  MoveL 6780 to (239.29, 155.73, 97.46) mm, rotated rx -180 ry 0 rz 180 deg; joints [-29.499, 18.299, 56.156, 64.652, 33.015, -60.536]
  Call Extruder(263.09151)
  MoveL 6781 to (239.16, 156.02, 97.46) mm, rotated rx 180 ry 0 rz -180 deg; joints [-29.531, 18.307, 56.146, 64.678, 33.044, -60.557]
  MoveL 6782 to (239.16, 156.02, 97.46) mm, rotated rx 180 ry 0 rz -180 deg; joints [-29.531, 18.307, 56.146, 64.678, 33.044, -60.557]
  Call Extruder(263.26194)
  MoveL 6783 to (239.05, 156.29, 97.46) mm, rotated rx 180 ry 0 rz 180 deg; joints [-29.561, 18.313, 56.137, 64.702, 33.071, -60.576]
  MoveL 6784 to (239.05, 156.29, 97.46) mm, rotated rx 180 ry 0 rz 180 deg; joints [-29.561, 18.313, 56.137, 64.702, 33.071, -60.576]
  Call Extruder(263.41995)
  MoveL 6785 to (238.94, 156.54, 97.46) mm, rotated rx -180 ry 0 rz 180 deg; joints [-29.589, 18.319, 56.129, 64.725, 33.096, -60.594]
  MoveL 6786 to (238.94, 156.54, 97.46) mm, rotated rx -180 ry 0 rz 180 deg; joints [-29.589, 18.319, 56.129, 64.725, 33.096, -60.594]
  Call Extruder(263.57856)
  MoveL 6787 to (238.84, 156.79, 97.46) mm, rotated rx 180 ry 0 rz 180 deg; joints [-29.617, 18.325, 56.121, 64.747, 33.121, -60.611]
  MoveL 6788 to (238.84, 156.79, 97.46) mm, rotated rx 180 ry 0 rz 180 deg; joints [-29.617, 18.325, 56.121, 64.747, 33.121, -60.611]
  Call Extruder(263.78473)
  MoveL 6789 to (238.66, 157.09, 97.46) mm, rotated rx -180 ry 0 rz 180 deg; joints [-29.653, 18.325, 56.121, 64.78, 33.153, -60.639]
  MoveL 6790 to (238.66, 157.09, 97.46) mm, rotated rx -180 ry 0 rz 180 deg; joints [-29.653, 18.325, 56.121, 64.78, 33.153, -60.639]
  Call Extruder(263.99168)
  MoveL 6791 to (238.49, 157.4, 97.46) mm, rotated rx 180 ry 0 rz 180 deg; joints [-29.689, 18.325, 56.122, 64.812, 33.184, -60.666]
  MoveL 6792 to (238.49, 157.4, 97.46) mm, rotated rx 180 ry 0 rz 180 deg; joints [-29.689, 18.325, 56.122, 64.812, 33.184, -60.666]
  Call Extruder(264.19941)
  MoveL 6793 to (238.31, 157.7, 97.46) mm, rotated rx -180 ry 0 rz -180 deg; joints [-29.725, 18.324, 56.122, 64.845, 33.216, -60.693]
  MoveL 6794 to (238.31, 157.7, 97.46) mm, rotated rx -180 ry 0 rz -180 deg; joints [-29.725, 18.324, 56.122, 64.845, 33.216, -60.693]
  Call Extruder(264.40791)
  MoveL 6795 to (238.13, 158.01, 97.46) mm, rotated rx 180 ry 0 rz 180 deg; joints [-29.761, 18.324, 56.123, 64.877, 33.247, -60.721]
  MoveL 6796 to (238.13, 158.01, 97.46) mm, rotated rx 180 ry 0 rz 180 deg; joints [-29.761, 18.324, 56.123, 64.877, 33.247, -60.721]
  Call Extruder(264.58745)
  MoveL 6797 to (237.96, 158.25, 97.46) mm, rotated rx 180 ry 0 rz 180 deg; joints [-29.792, 18.318, 56.131, 64.907, 33.273, -60.747]
  MoveL 6798 to (237.96, 158.25, 97.46) mm, rotated rx 180 ry 0 rz 180 deg; joints [-29.792, 18.318, 56.131, 64.907, 33.273, -60.747]
  Call Extruder(264.92086)
  MoveL 6799 to (237.63, 158.7, 97.46) mm, rotated rx -180 ry 0 rz 180 deg; joints [-29.849, 18.306, 56.147, 64.963, 33.322, -60.796]
  MoveL 6800 to (237.63, 158.7, 97.46) mm, rotated rx -180 ry 0 rz 180 deg; joints [-29.849, 18.306, 56.147, 64.963, 33.322, -60.796]
  Call Extruder(265.25545)
  MoveL 6801 to (237.3, 159.15, 97.46) mm, rotated rx 180 ry 0 rz 180 deg; joints [-29.907, 18.294, 56.162, 65.019, 33.37, -60.844]
  Call Extruder(266.08341)
  MoveL 6802 to (236.39, 160.19, 97.46) mm, rotated rx 180 ry 0 rz -180 deg; joints [-30.046, 18.239, 56.234, 65.166, 33.485, -60.975]
  Call Extruder(266.91134)
  MoveL 6803 to (235.35, 161.1, 97.46) mm, rotated rx 180 ry 0 rz 180 deg; joints [-30.182, 18.151, 56.349, 65.322, 33.592, -61.119]
  Call Extruder(267.07865)
  MoveL 6804 to (235.13, 161.27, 97.46) mm, rotated rx 180 ry 0 rz 180 deg; joints [-30.208, 18.129, 56.379, 65.355, 33.612, -61.15]
  MoveL 6805 to (235.13, 161.27, 97.46) mm, rotated rx 180 ry 0 rz 180 deg; joints [-30.208, 18.129, 56.379, 65.355, 33.612, -61.15]
  Call Extruder(267.41207)
  MoveL 6806 to (234.68, 161.59, 97.46) mm, rotated rx 180 ry 0 rz 180 deg; joints [-30.261, 18.084, 56.438, 65.419, 33.652, -61.211]
  MoveL 6807 to (234.68, 161.59, 97.46) mm, rotated rx 180 ry 0 rz 180 deg; joints [-30.261, 18.084, 56.438, 65.419, 33.652, -61.211]
  Call Extruder(267.74432)
  MoveL 6808 to (234.23, 161.92, 97.46) mm, rotated rx 180 ry 0 rz 180 deg; joints [-30.314, 18.039, 56.497, 65.484, 33.693, -61.271]
  MoveL 6809 to (234.23, 161.92, 97.46) mm, rotated rx 180 ry 0 rz 180 deg; joints [-30.314, 18.039, 56.497, 65.484, 33.693, -61.271]
  Call Extruder(267.86197)
  MoveL 6810 to (234.05, 162.02, 97.46) mm, rotated rx 180 ry 0 rz 180 deg; joints [-30.331, 18.019, 56.522, 65.508, 33.706, -61.294]
  MoveL 6811 to (234.05, 162.02, 97.46) mm, rotated rx 180 ry 0 rz 180 deg; joints [-30.331, 18.019, 56.522, 65.508, 33.706, -61.294]
  Call Extruder(268.06970)
  MoveL 6812 to (233.75, 162.2, 97.46) mm, rotated rx 180 ry 0 rz 180 deg; joints [-30.363, 17.985, 56.567, 65.55, 33.729, -61.334]
  MoveL 6813 to (233.75, 162.2, 97.46) mm, rotated rx 180 ry 0 rz 180 deg; joints [-30.363, 17.985, 56.567, 65.55, 33.729, -61.334]
  Call Extruder(268.27665)
  MoveL 6814 to (233.45, 162.37, 97.46) mm, rotated rx 180 ry 0 rz 180 deg; joints [-30.394, 17.95, 56.613, 65.591, 33.753, -61.374]
  MoveL 6815 to (233.45, 162.37, 97.46) mm, rotated rx 180 ry 0 rz 180 deg; joints [-30.394, 17.95, 56.613, 65.591, 33.753, -61.374]
  Call Extruder(268.48282)
  MoveL 6816 to (233.14, 162.55, 97.46) mm, rotated rx 180 ry 0 rz 180 deg; joints [-30.426, 17.916, 56.658, 65.633, 33.776, -61.414]
  MoveL 6817 to (233.14, 162.55, 97.46) mm, rotated rx 180 ry 0 rz 180 deg; joints [-30.426, 17.916, 56.658, 65.633, 33.776, -61.414]
  Call Extruder(268.66449)
  MoveL 6818 to (232.87, 162.69, 97.46) mm, rotated rx -180 ry 0 rz 180 deg; joints [-30.453, 17.882, 56.701, 65.67, 33.796, -61.45]
  MoveL 6819 to (232.87, 162.69, 97.46) mm, rotated rx -180 ry 0 rz 180 deg; joints [-30.453, 17.882, 56.701, 65.67, 33.796, -61.45]
  Call Extruder(268.82246)
  MoveL 6820 to (232.62, 162.8, 97.46) mm, rotated rx -180 ry 0 rz 180 deg; joints [-30.476, 17.85, 56.743, 65.703, 33.811, -61.483]
  MoveL 6821 to (232.62, 162.8, 97.46) mm, rotated rx -180 ry 0 rz 180 deg; joints [-30.476, 17.85, 56.743, 65.703, 33.811, -61.483]
  Call Extruder(268.97983)
  MoveL 6822 to (232.37, 162.9, 97.46) mm, rotated rx 180 ry 0 rz 180 deg; joints [-30.498, 17.819, 56.784, 65.736, 33.827, -61.515]
  MoveL 6823 to (232.37, 162.9, 97.46) mm, rotated rx 180 ry 0 rz 180 deg; joints [-30.498, 17.819, 56.784, 65.736, 33.827, -61.515]
  Call Extruder(269.16257)
  MoveL 6824 to (232.08, 163.02, 97.46) mm, rotated rx 180 ry 0 rz 180 deg; joints [-30.524, 17.781, 56.834, 65.774, 33.846, -61.552]
  MoveL 6825 to (232.08, 163.02, 97.46) mm, rotated rx 180 ry 0 rz 180 deg; joints [-30.524, 17.781, 56.834, 65.774, 33.846, -61.552]
  Call Extruder(269.34456)
  MoveL 6826 to (231.78, 163.15, 97.46) mm, rotated rx -180 ry 0 rz 180 deg; joints [-30.551, 17.743, 56.883, 65.812, 33.864, -61.589]
  MoveL 6827 to (231.78, 163.15, 97.46) mm, rotated rx -180 ry 0 rz 180 deg; joints [-30.551, 17.743, 56.883, 65.812, 33.864, -61.589]
  Call Extruder(269.49190)
  MoveL 6828 to (231.54, 163.24, 97.46) mm, rotated rx 180 ry 0 rz 180 deg; joints [-30.571, 17.711, 56.924, 65.842, 33.878, -61.62]
  MoveL 6829 to (231.54, 163.24, 97.46) mm, rotated rx 180 ry 0 rz 180 deg; joints [-30.571, 17.711, 56.924, 65.842, 33.878, -61.62]
  Call Extruder(269.60512)
  MoveL 6830 to (231.35, 163.3, 97.46) mm, rotated rx 180 ry 0 rz 180 deg; joints [-30.587, 17.685, 56.958, 65.866, 33.889, -61.644]
  MoveL 6831 to (231.35, 163.3, 97.46) mm, rotated rx 180 ry 0 rz 180 deg; joints [-30.587, 17.685, 56.958, 65.866, 33.889, -61.644]
  Call Extruder(269.71789)
  MoveL 6832 to (231.17, 163.36, 97.46) mm, rotated rx 180 ry 0 rz 180 deg; joints [-30.602, 17.659, 56.992, 65.89, 33.899, -61.667]
  MoveL 6833 to (231.17, 163.36, 97.46) mm, rotated rx 180 ry 0 rz 180 deg; joints [-30.602, 17.659, 56.992, 65.89, 33.899, -61.667]
  Call Extruder(269.83022)
  MoveL 6834 to (230.98, 163.42, 97.46) mm, rotated rx 180 ry 0 rz -180 deg; joints [-30.618, 17.633, 57.026, 65.914, 33.909, -61.691]
  MoveL 6835 to (230.98, 163.42, 97.46) mm, rotated rx 180 ry 0 rz -180 deg; joints [-30.618, 17.633, 57.026, 65.914, 33.909, -61.691]
  Call Extruder(269.94211)
  MoveL 6836 to (230.79, 163.48, 97.46) mm, rotated rx 180 ry 0 rz 180 deg; joints [-30.633, 17.607, 57.06, 65.937, 33.92, -61.715]
  MoveL 6837 to (230.79, 163.48, 97.46) mm, rotated rx 180 ry 0 rz 180 deg; joints [-30.633, 17.607, 57.06, 65.937, 33.92, -61.715]
  Call Extruder(270.06351)
  MoveL 6838 to (230.58, 163.55, 97.46) mm, rotated rx 180 ry 0 rz 180 deg; joints [-30.65, 17.579, 57.097, 65.963, 33.931, -61.74]
  MoveL 6839 to (230.58, 163.55, 97.46) mm, rotated rx 180 ry 0 rz 180 deg; joints [-30.65, 17.579, 57.097, 65.963, 33.931, -61.74]
  Call Extruder(270.19433)
  MoveL 6840 to (230.36, 163.62, 97.46) mm, rotated rx 180 ry 0 rz 180 deg; joints [-30.668, 17.548, 57.137, 65.991, 33.943, -61.768]
  MoveL 6841 to (230.36, 163.62, 97.46) mm, rotated rx 180 ry 0 rz 180 deg; joints [-30.668, 17.548, 57.137, 65.991, 33.943, -61.768]
  Call Extruder(270.32458)
  MoveL 6842 to (230.14, 163.68, 97.46) mm, rotated rx 180 ry 0 rz 180 deg; joints [-30.685, 17.516, 57.178, 66.019, 33.955, -61.796]
  MoveL 6843 to (230.14, 163.68, 97.46) mm, rotated rx 180 ry 0 rz 180 deg; joints [-30.685, 17.516, 57.178, 66.019, 33.955, -61.796]
  Call Extruder(270.45426)
  MoveL 6844 to (229.91, 163.75, 97.46) mm, rotated rx 180 ry 0 rz 180 deg; joints [-30.703, 17.485, 57.218, 66.047, 33.967, -61.824]
  MoveL 6845 to (229.91, 163.75, 97.46) mm, rotated rx 180 ry 0 rz 180 deg; joints [-30.703, 17.485, 57.218, 66.047, 33.967, -61.824]
  Call Extruder(270.58338)
  MoveL 6846 to (229.69, 163.82, 97.46) mm, rotated rx -180 ry 0 rz -180 deg; joints [-30.721, 17.454, 57.259, 66.074, 33.979, -61.852]
  MoveL 6847 to (229.69, 163.82, 97.46) mm, rotated rx -180 ry 0 rz -180 deg; joints [-30.721, 17.454, 57.259, 66.074, 33.979, -61.852]
  Call Extruder(270.69845)
  MoveL 6848 to (229.48, 163.86, 97.46) mm, rotated rx -180 ry 0 rz -180 deg; joints [-30.736, 17.424, 57.298, 66.099, 33.988, -61.877]
  MoveL 6849 to (229.48, 163.86, 97.46) mm, rotated rx -180 ry 0 rz -180 deg; joints [-30.736, 17.424, 57.298, 66.099, 33.988, -61.877]
  Call Extruder(270.81308)
  MoveL 6850 to (229.28, 163.91, 97.46) mm, rotated rx 180 ry 0 rz 180 deg; joints [-30.751, 17.394, 57.337, 66.124, 33.998, -61.902]
  MoveL 6851 to (229.28, 163.91, 97.46) mm, rotated rx 180 ry 0 rz 180 deg; joints [-30.751, 17.394, 57.337, 66.124, 33.998, -61.902]
  Call Extruder(270.92725)
  MoveL 6852 to (229.08, 163.95, 97.46) mm, rotated rx 180 ry 0 rz 180 deg; joints [-30.766, 17.364, 57.376, 66.148, 34.007, -61.927]
  MoveL 6853 to (229.08, 163.95, 97.46) mm, rotated rx 180 ry 0 rz 180 deg; joints [-30.766, 17.364, 57.376, 66.148, 34.007, -61.927]
  Call Extruder(271.04096)
  MoveL 6854 to (228.87, 164, 97.46) mm, rotated rx -180 ry 0 rz 180 deg; joints [-30.781, 17.334, 57.415, 66.173, 34.017, -61.952]
  MoveL 6855 to (228.87, 164, 97.46) mm, rotated rx -180 ry 0 rz 180 deg; joints [-30.781, 17.334, 57.415, 66.173, 34.017, -61.952]
  Call Extruder(271.16638)
  MoveL 6856 to (228.64, 164.04, 97.46) mm, rotated rx -180 ry 0 rz 180 deg; joints [-30.797, 17.3, 57.458, 66.2, 34.027, -61.979]
  MoveL 6857 to (228.64, 164.04, 97.46) mm, rotated rx -180 ry 0 rz 180 deg; joints [-30.797, 17.3, 57.458, 66.2, 34.027, -61.979]
  Call Extruder(271.30336)
  MoveL 6858 to (228.4, 164.09, 97.46) mm, rotated rx 180 ry 0 rz 180 deg; joints [-30.815, 17.263, 57.506, 66.23, 34.038, -62.01]
  MoveL 6859 to (228.4, 164.09, 97.46) mm, rotated rx 180 ry 0 rz 180 deg; joints [-30.815, 17.263, 57.506, 66.23, 34.038, -62.01]
  Call Extruder(271.43973)
  MoveL 6860 to (228.15, 164.14, 97.46) mm, rotated rx 180 ry 0 rz 180 deg; joints [-30.832, 17.226, 57.555, 66.259, 34.05, -62.04]
  MoveL 6861 to (228.15, 164.14, 97.46) mm, rotated rx 180 ry 0 rz 180 deg; joints [-30.832, 17.226, 57.555, 66.259, 34.05, -62.04]
  Call Extruder(271.57549)
  MoveL 6862 to (227.9, 164.19, 97.46) mm, rotated rx -180 ry 0 rz 180 deg; joints [-30.85, 17.189, 57.602, 66.289, 34.061, -62.07]
  MoveL 6863 to (227.9, 164.19, 97.46) mm, rotated rx -180 ry 0 rz 180 deg; joints [-30.85, 17.189, 57.602, 66.289, 34.061, -62.07]
  Call Extruder(271.71064)
  MoveL 6864 to (227.65, 164.24, 97.46) mm, rotated rx 180 ry 0 rz 180 deg; joints [-30.868, 17.152, 57.65, 66.319, 34.072, -62.1]
  MoveL 6865 to (227.65, 164.24, 97.46) mm, rotated rx 180 ry 0 rz 180 deg; joints [-30.868, 17.152, 57.65, 66.319, 34.072, -62.1]
  Call Extruder(271.84517)
  MoveL 6866 to (227.4, 164.29, 97.46) mm, rotated rx 180 ry 0 rz 180 deg; joints [-30.886, 17.115, 57.698, 66.348, 34.083, -62.13]
  MoveL 6867 to (227.4, 164.29, 97.46) mm, rotated rx 180 ry 0 rz 180 deg; joints [-30.886, 17.115, 57.698, 66.348, 34.083, -62.13]
  Call Extruder(271.97910)
  MoveL 6868 to (227.15, 164.34, 97.46) mm, rotated rx 180 ry 0 rz 180 deg; joints [-30.903, 17.078, 57.746, 66.377, 34.095, -62.16]
  MoveL 6869 to (227.15, 164.34, 97.46) mm, rotated rx 180 ry 0 rz 180 deg; joints [-30.903, 17.078, 57.746, 66.377, 34.095, -62.16]
  Call Extruder(272.12696)
  MoveL 6870 to (226.87, 164.39, 97.46) mm, rotated rx 180 ry 0 rz 180 deg; joints [-30.923, 17.037, 57.799, 66.41, 34.107, -62.193]
  MoveL 6871 to (226.87, 164.39, 97.46) mm, rotated rx 180 ry 0 rz 180 deg; joints [-30.923, 17.037, 57.799, 66.41, 34.107, -62.193]
  Call Extruder(272.28870)
  MoveL 6872 to (226.57, 164.44, 97.46) mm, rotated rx 180 ry 0 rz 180 deg; joints [-30.943, 16.99, 57.859, 66.445, 34.12, -62.229]
  MoveL 6873 to (226.57, 164.44, 97.46) mm, rotated rx 180 ry 0 rz 180 deg; joints [-30.943, 16.99, 57.859, 66.445, 34.12, -62.229]
  Call Extruder(272.44972)
  MoveL 6874 to (226.26, 164.49, 97.46) mm, rotated rx 180 ry 0 rz 180 deg; joints [-30.964, 16.944, 57.919, 66.481, 34.133, -62.265]
  MoveL 6875 to (226.26, 164.49, 97.46) mm, rotated rx 180 ry 0 rz 180 deg; joints [-30.964, 16.944, 57.919, 66.481, 34.133, -62.265]
  Call Extruder(272.61000)
  MoveL 6876 to (225.96, 164.54, 97.46) mm, rotated rx 180 ry 0 rz 180 deg; joints [-30.985, 16.897, 57.979, 66.516, 34.146, -62.301]
  MoveL 6877 to (225.96, 164.54, 97.46) mm, rotated rx 180 ry 0 rz 180 deg; joints [-30.985, 16.897, 57.979, 66.516, 34.146, -62.301]
  Call Extruder(272.76956)
  MoveL 6878 to (225.65, 164.58, 97.46) mm, rotated rx 180 ry 0 rz 180 deg; joints [-31.006, 16.851, 58.038, 66.551, 34.159, -62.337]
  MoveL 6879 to (225.65, 164.58, 97.46) mm, rotated rx 180 ry 0 rz 180 deg; joints [-31.006, 16.851, 58.038, 66.551, 34.159, -62.337]
  Call Extruder(272.92838)
  MoveL 6880 to (225.34, 164.63, 97.46) mm, rotated rx 180 ry 0 rz 180 deg; joints [-31.027, 16.805, 58.098, 66.586, 34.172, -62.373]
  MoveL 6881 to (225.34, 164.63, 97.46) mm, rotated rx 180 ry 0 rz 180 deg; joints [-31.027, 16.805, 58.098, 66.586, 34.172, -62.373]
  Call Extruder(273.10706)
  MoveL 6882 to (225, 164.68, 97.46) mm, rotated rx 180 ry 0 rz 180 deg; joints [-31.049, 16.752, 58.166, 66.626, 34.187, -62.414]
  MoveL 6883 to (225, 164.68, 97.46) mm, rotated rx 180 ry 0 rz 180 deg; joints [-31.049, 16.752, 58.166, 66.626, 34.187, -62.414]
  Call Extruder(273.30550)
  MoveL 6884 to (224.61, 164.73, 97.46) mm, rotated rx -180 ry 0 rz -180 deg; joints [-31.074, 16.692, 58.243, 66.67, 34.202, -62.459]
  MoveL 6885 to (224.61, 164.73, 97.46) mm, rotated rx -180 ry 0 rz -180 deg; joints [-31.074, 16.692, 58.243, 66.67, 34.202, -62.459]
  Call Extruder(273.50307)
  MoveL 6886 to (224.22, 164.77, 97.46) mm, rotated rx 180 ry 0 rz 180 deg; joints [-31.1, 16.632, 58.32, 66.713, 34.217, -62.504]
  MoveL 6887 to (224.22, 164.77, 97.46) mm, rotated rx 180 ry 0 rz 180 deg; joints [-31.1, 16.632, 58.32, 66.713, 34.217, -62.504]
  Call Extruder(273.69978)
  MoveL 6888 to (223.84, 164.82, 97.46) mm, rotated rx 180 ry 0 rz 180 deg; joints [-31.125, 16.573, 58.397, 66.757, 34.233, -62.548]
  MoveL 6889 to (223.84, 164.82, 97.46) mm, rotated rx 180 ry 0 rz 180 deg; joints [-31.125, 16.573, 58.397, 66.757, 34.233, -62.548]
  Call Extruder(273.89562)
  MoveL 6890 to (223.45, 164.86, 97.46) mm, rotated rx 180 ry 0 rz 180 deg; joints [-31.15, 16.513, 58.473, 66.8, 34.249, -62.593]
  MoveL 6891 to (223.45, 164.86, 97.46) mm, rotated rx 180 ry 0 rz 180 deg; joints [-31.15, 16.513, 58.473, 66.8, 34.249, -62.593]
  Call Extruder(274.19098)
  MoveL 6892 to (222.86, 164.91, 97.46) mm, rotated rx -180 ry 0 rz 180 deg; joints [-31.186, 16.42, 58.592, 66.865, 34.27, -62.66]
  MoveL 6893 to (222.86, 164.91, 97.46) mm, rotated rx -180 ry 0 rz 180 deg; joints [-31.186, 16.42, 58.592, 66.865, 34.27, -62.66]
  Call Extruder(274.48500)
  MoveL 6894 to (222.27, 164.95, 97.46) mm, rotated rx -180 ry 0 rz 180 deg; joints [-31.222, 16.327, 58.711, 66.929, 34.292, -62.727]
  MoveL 6895 to (222.27, 164.95, 97.46) mm, rotated rx -180 ry 0 rz 180 deg; joints [-31.222, 16.327, 58.711, 66.929, 34.292, -62.727]
  Call Extruder(274.77770)
  MoveL 6896 to (221.68, 165, 97.46) mm, rotated rx 180 ry 0 rz 180 deg; joints [-31.258, 16.235, 58.829, 66.993, 34.315, -62.793]
  MoveL 6897 to (221.68, 165, 97.46) mm, rotated rx 180 ry 0 rz 180 deg; joints [-31.258, 16.235, 58.829, 66.993, 34.315, -62.793]
  Call Extruder(275.35114)
  MoveL 6898 to (220.52, 165.05, 97.46) mm, rotated rx 180 ry 0 rz 180 deg; joints [-31.326, 16.048, 59.067, 67.117, 34.355, -62.922]
  MoveL 6899 to (220.52, 165.05, 97.46) mm, rotated rx 180 ry 0 rz 180 deg; joints [-31.326, 16.048, 59.067, 67.117, 34.355, -62.922]
  Call Extruder(276.06515)
  MoveL 6900 to (219.06, 165.09, 97.46) mm, rotated rx 180 ry 0 rz 180 deg; joints [-31.409, 15.814, 59.365, 67.27, 34.404, -63.081]
  Call Extruder(392.91189)
  MoveL 6901 to (-19.06, 165.09, 97.46) mm, rotated rx 180 ry 0 rz 180 deg; joints [-51.475, -13.284, 89.091, 78.954, 52.855, -72.085]
  Call Extruder(393.34049)
  MoveL 6902 to (-19.94, 165.07, 97.46) mm, rotated rx -180 ry 0 rz 180 deg; joints [-51.582, -13.365, 89.153, 78.982, 52.96, -72.087]
  MoveL 6903 to (-19.94, 165.07, 97.46) mm, rotated rx -180 ry 0 rz 180 deg; joints [-51.582, -13.365, 89.153, 78.982, 52.96, -72.087]
  Call Extruder(393.91395)
  MoveL 6904 to (-21.1, 165.03, 97.46) mm, rotated rx 180 ry 0 rz -180 deg; joints [-51.722, -13.474, 89.237, 79.017, 53.098, -72.089]
  MoveL 6905 to (-21.1, 165.03, 97.46) mm, rotated rx 180 ry 0 rz -180 deg; joints [-51.722, -13.474, 89.237, 79.017, 53.098, -72.089]
  Call Extruder(394.34824)
  MoveL 6906 to (-21.97, 164.98, 97.46) mm, rotated rx 180 ry 0 rz 180 deg; joints [-51.827, -13.557, 89.301, 79.044, 53.201, -72.09]
  MoveL 6907 to (-21.97, 164.98, 97.46) mm, rotated rx 180 ry 0 rz 180 deg; joints [-51.827, -13.557, 89.301, 79.044, 53.201, -72.09]
  Call Extruder(394.64227)
  MoveL 6908 to (-22.56, 164.93, 97.46) mm, rotated rx 180 ry 0 rz -180 deg; joints [-51.897, -13.615, 89.345, 79.06, 53.27, -72.089]
  MoveL 6909 to (-22.56, 164.93, 97.46) mm, rotated rx 180 ry 0 rz -180 deg; joints [-51.897, -13.615, 89.345, 79.06, 53.27, -72.089]
  Call Extruder(394.93763)
  MoveL 6910 to (-23.15, 164.89, 97.46) mm, rotated rx 180 ry 0 rz 180 deg; joints [-51.966, -13.672, 89.39, 79.077, 53.339, -72.089]
  MoveL 6911 to (-23.15, 164.89, 97.46) mm, rotated rx 180 ry 0 rz 180 deg; joints [-51.966, -13.672, 89.39, 79.077, 53.339, -72.089]
  Call Extruder(395.18385)
  MoveL 6912 to (-23.64, 164.84, 97.46) mm, rotated rx 180 ry 0 rz 180 deg; joints [-52.023, -13.721, 89.427, 79.091, 53.395, -72.088]
  MoveL 6913 to (-23.64, 164.84, 97.46) mm, rotated rx 180 ry 0 rz 180 deg; joints [-52.023, -13.721, 89.427, 79.091, 53.395, -72.088]
  Call Extruder(395.38056)
  MoveL 6914 to (-24.03, 164.79, 97.46) mm, rotated rx 180 ry 0 rz 180 deg; joints [-52.067, -13.76, 89.457, 79.101, 53.439, -72.087]
  MoveL 6915 to (-24.03, 164.79, 97.46) mm, rotated rx 180 ry 0 rz 180 deg; joints [-52.067, -13.76, 89.457, 79.101, 53.439, -72.087]
  Call Extruder(395.57813)
  MoveL 6916 to (-24.42, 164.75, 97.46) mm, rotated rx -180 ry 0 rz 180 deg; joints [-52.112, -13.8, 89.487, 79.111, 53.483, -72.085]
  MoveL 6917 to (-24.42, 164.75, 97.46) mm, rotated rx -180 ry 0 rz 180 deg; joints [-52.112, -13.8, 89.487, 79.111, 53.483, -72.085]
  Call Extruder(395.77657)
  MoveL 6918 to (-24.8, 164.7, 97.46) mm, rotated rx -180 ry 0 rz 180 deg; joints [-52.156, -13.839, 89.517, 79.121, 53.527, -72.084]
  MoveL 6919 to (-24.8, 164.7, 97.46) mm, rotated rx -180 ry 0 rz 180 deg; joints [-52.156, -13.839, 89.517, 79.121, 53.527, -72.084]
  Call Extruder(395.97588)
  MoveL 6920 to (-25.19, 164.66, 97.46) mm, rotated rx 180 ry 0 rz 180 deg; joints [-52.2, -13.878, 89.547, 79.132, 53.571, -72.083]
  MoveL 6921 to (-25.19, 164.66, 97.46) mm, rotated rx 180 ry 0 rz 180 deg; joints [-52.2, -13.878, 89.547, 79.132, 53.571, -72.083]
  Call Extruder(396.13471)
  MoveL 6922 to (-25.5, 164.61, 97.46) mm, rotated rx 180 ry 0 rz 180 deg; joints [-52.235, -13.911, 89.572, 79.139, 53.605, -72.081]
  MoveL 6923 to (-25.5, 164.61, 97.46) mm, rotated rx 180 ry 0 rz 180 deg; joints [-52.235, -13.911, 89.572, 79.139, 53.605, -72.081]
  Call Extruder(396.29427)
  MoveL 6924 to (-25.8, 164.56, 97.46) mm, rotated rx 180 ry 0 rz 180 deg; joints [-52.269, -13.943, 89.597, 79.147, 53.639, -72.08]
  MoveL 6925 to (-25.8, 164.56, 97.46) mm, rotated rx 180 ry 0 rz 180 deg; joints [-52.269, -13.943, 89.597, 79.147, 53.639, -72.08]
  Call Extruder(396.45456)
  MoveL 6926 to (-26.11, 164.51, 97.46) mm, rotated rx 180 ry 0 rz -180 deg; joints [-52.303, -13.976, 89.621, 79.154, 53.672, -72.078]
  MoveL 6927 to (-26.11, 164.51, 97.46) mm, rotated rx 180 ry 0 rz -180 deg; joints [-52.303, -13.976, 89.621, 79.154, 53.672, -72.078]
  Call Extruder(396.61557)
  MoveL 6928 to (-26.41, 164.46, 97.46) mm, rotated rx 180 ry 0 rz -180 deg; joints [-52.337, -14.008, 89.646, 79.161, 53.706, -72.076]
  MoveL 6929 to (-26.41, 164.46, 97.46) mm, rotated rx 180 ry 0 rz -180 deg; joints [-52.337, -14.008, 89.646, 79.161, 53.706, -72.076]
  Call Extruder(396.77732)
  MoveL 6930 to (-26.72, 164.41, 97.46) mm, rotated rx 180 ry 0 rz 180 deg; joints [-52.371, -14.04, 89.671, 79.169, 53.74, -72.075]
  MoveL 6931 to (-26.72, 164.41, 97.46) mm, rotated rx 180 ry 0 rz 180 deg; joints [-52.371, -14.04, 89.671, 79.169, 53.74, -72.075]
  Call Extruder(396.93979)
  MoveL 6932 to (-27.02, 164.37, 97.46) mm, rotated rx 180 ry 0 rz 180 deg; joints [-52.405, -14.073, 89.695, 79.176, 53.774, -72.073]
  MoveL 6933 to (-27.02, 164.37, 97.46) mm, rotated rx 180 ry 0 rz 180 deg; joints [-52.405, -14.073, 89.695, 79.176, 53.774, -72.073]
  Call Extruder(397.07371)
  MoveL 6934 to (-27.27, 164.32, 97.46) mm, rotated rx -180 ry 0 rz -180 deg; joints [-52.432, -14.1, 89.716, 79.182, 53.801, -72.071]
  MoveL 6935 to (-27.27, 164.32, 97.46) mm, rotated rx -180 ry 0 rz -180 deg; joints [-52.432, -14.1, 89.716, 79.182, 53.801, -72.071]
  Call Extruder(397.20825)
  MoveL 6936 to (-27.52, 164.27, 97.46) mm, rotated rx 180 ry 0 rz 180 deg; joints [-52.459, -14.127, 89.737, 79.187, 53.828, -72.069]
  MoveL 6937 to (-27.52, 164.27, 97.46) mm, rotated rx 180 ry 0 rz 180 deg; joints [-52.459, -14.127, 89.737, 79.187, 53.828, -72.069]
  Call Extruder(397.34340)
  MoveL 6938 to (-27.77, 164.22, 97.46) mm, rotated rx 180 ry 0 rz 180 deg; joints [-52.486, -14.155, 89.758, 79.193, 53.855, -72.067]
  MoveL 6939 to (-27.77, 164.22, 97.46) mm, rotated rx 180 ry 0 rz 180 deg; joints [-52.486, -14.155, 89.758, 79.193, 53.855, -72.067]
  Call Extruder(397.47915)
  MoveL 6940 to (-28.02, 164.17, 97.46) mm, rotated rx 180 ry 0 rz -180 deg; joints [-52.513, -14.182, 89.779, 79.199, 53.882, -72.065]
  MoveL 6941 to (-28.02, 164.17, 97.46) mm, rotated rx 180 ry 0 rz -180 deg; joints [-52.513, -14.182, 89.779, 79.199, 53.882, -72.065]
  Call Extruder(397.61552)
  MoveL 6942 to (-28.27, 164.12, 97.46) mm, rotated rx 180 ry 0 rz 180 deg; joints [-52.54, -14.21, 89.799, 79.204, 53.909, -72.063]
  MoveL 6943 to (-28.27, 164.12, 97.46) mm, rotated rx 180 ry 0 rz 180 deg; joints [-52.54, -14.21, 89.799, 79.204, 53.909, -72.063]
  Call Extruder(397.70039)
  MoveL 6944 to (-28.43, 164.09, 97.46) mm, rotated rx 180 ry 0 rz -180 deg; joints [-52.556, -14.227, 89.812, 79.208, 53.925, -72.062]
  Set speed (130.0 mm/s)
  MoveL 6945 to (-31.76, 163.31, 97.46) mm, rotated rx 180 ry 0 rz 180 deg; joints [-52.91, -14.605, 90.097, 79.276, 54.279, -72.028]
  MoveL 6946 to (-31.76, 163.31, 106.87) mm, rotated rx 180 ry 0 rz 180 deg; joints [-52.91, -15.274, 92.047, 80.186, 54.05, -73.582]
  Call Extruder(395.70039)
  Set speed (40.0 mm/s)
  MoveL 6947 to (-31.76, 163.31, 106.87) mm, rotated rx 180 ry 0 rz 180 deg; joints [-52.91, -15.274, 92.047, 80.186, 54.05, -73.582]
  Call Extruder(0.00000)
  Set speed (130.0 mm/s)
  MoveL 6948 to (-31.64, 163.21, 106.87) mm, rotated rx 180 ry 0 rz 180 deg; joints [-52.884, -15.275, 92.048, 80.177, 54.026, -73.576]
  Call Extruder(2.00000)
  Set speed (40.0 mm/s)
  MoveL 6949 to (-31.64, 163.21, 106.87) mm, rotated rx 180 ry 0 rz 180 deg; joints [-52.884, -15.275, 92.048, 80.177, 54.026, -73.576]
  Set speed (30.0 mm/s)
  MoveL 6950 to (-31.64, 163.21, 106.87) mm, rotated rx 180 ry 0 rz 180 deg; joints [-52.884, -15.275, 92.048, 80.177, 54.026, -73.576]
  Call Extruder(2.18198)
  MoveL 6951 to (-31.93, 163.09, 106.87) mm, rotated rx 180 ry 0 rz 180 deg; joints [-52.91, -15.315, 92.077, 80.179, 54.052, -73.57]
  MoveL 6952 to (-31.93, 163.09, 106.87) mm, rotated rx 180 ry 0 rz 180 deg; joints [-52.91, -15.315, 92.077, 80.179, 54.052, -73.57]
  Call Extruder(2.36471)
  MoveL 6953 to (-32.22, 162.97, 106.87) mm, rotated rx -180 ry 0 rz -180 deg; joints [-52.936, -15.354, 92.106, 80.18, 54.079, -73.563]
  MoveL 6954 to (-32.22, 162.97, 106.87) mm, rotated rx -180 ry 0 rz -180 deg; joints [-52.936, -15.354, 92.106, 80.18, 54.079, -73.563]
  Call Extruder(2.53513)
  MoveL 6955 to (-32.49, 162.85, 106.87) mm, rotated rx 180 ry 0 rz 180 deg; joints [-52.96, -15.39, 92.133, 80.182, 54.104, -73.556]
  MoveL 6956 to (-32.49, 162.85, 106.87) mm, rotated rx 180 ry 0 rz 180 deg; joints [-52.96, -15.39, 92.133, 80.182, 54.104, -73.556]
  Call Extruder(2.69310)
  MoveL 6957 to (-32.74, 162.74, 106.87) mm, rotated rx -180 ry 0 rz 180 deg; joints [-52.982, -15.424, 92.159, 80.183, 54.126, -73.55]
  MoveL 6958 to (-32.74, 162.74, 106.87) mm, rotated rx -180 ry 0 rz 180 deg; joints [-52.982, -15.424, 92.159, 80.183, 54.126, -73.55]
  Call Extruder(2.85168)
  MoveL 6959 to (-32.99, 162.64, 106.87) mm, rotated rx 180 ry 0 rz -180 deg; joints [-53.004, -15.458, 92.184, 80.185, 54.149, -73.544]
  MoveL 6960 to (-32.99, 162.64, 106.87) mm, rotated rx 180 ry 0 rz -180 deg; joints [-53.004, -15.458, 92.184, 80.185, 54.149, -73.544]
  Call Extruder(3.05785)
  MoveL 6961 to (-33.29, 162.46, 106.87) mm, rotated rx 180 ry 0 rz 180 deg; joints [-53.026, -15.504, 92.218, 80.184, 54.172, -73.533]
  MoveL 6962 to (-33.29, 162.46, 106.87) mm, rotated rx 180 ry 0 rz 180 deg; joints [-53.026, -15.504, 92.218, 80.184, 54.172, -73.533]
  Call Extruder(3.26479)
  MoveL 6963 to (-33.6, 162.29, 106.87) mm, rotated rx -180 ry 0 rz 180 deg; joints [-53.049, -15.551, 92.252, 80.183, 54.196, -73.523]
  MoveL 6964 to (-33.6, 162.29, 106.87) mm, rotated rx -180 ry 0 rz 180 deg; joints [-53.049, -15.551, 92.252, 80.183, 54.196, -73.523]
  Call Extruder(3.47251)
  MoveL 6965 to (-33.9, 162.11, 106.87) mm, rotated rx 180 ry 0 rz 180 deg; joints [-53.071, -15.597, 92.286, 80.183, 54.22, -73.513]
  MoveL 6966 to (-33.9, 162.11, 106.87) mm, rotated rx 180 ry 0 rz 180 deg; joints [-53.071, -15.597, 92.286, 80.183, 54.22, -73.513]
  Call Extruder(3.68101)
  MoveL 6967 to (-34.21, 161.94, 106.87) mm, rotated rx 180 ry 0 rz 180 deg; joints [-53.094, -15.644, 92.32, 80.182, 54.243, -73.503]
  MoveL 6968 to (-34.21, 161.94, 106.87) mm, rotated rx 180 ry 0 rz 180 deg; joints [-53.094, -15.644, 92.32, 80.182, 54.243, -73.503]
  Call Extruder(3.86055)
  MoveL 6969 to (-34.45, 161.76, 106.87) mm, rotated rx -180 ry 0 rz 180 deg; joints [-53.109, -15.685, 92.351, 80.179, 54.259, -73.493]
  MoveL 6970 to (-34.45, 161.76, 106.87) mm, rotated rx -180 ry 0 rz 180 deg; joints [-53.109, -15.685, 92.351, 80.179, 54.259, -73.493]
  Call Extruder(4.19399)
  MoveL 6971 to (-34.9, 161.43, 106.87) mm, rotated rx 180 ry 0 rz 180 deg; joints [-53.135, -15.761, 92.407, 80.174, 54.289, -73.474]
  MoveL 6972 to (-34.9, 161.43, 106.87) mm, rotated rx 180 ry 0 rz 180 deg; joints [-53.135, -15.761, 92.407, 80.174, 54.289, -73.474]
  Call Extruder(4.52861)
  MoveL 6973 to (-35.35, 161.1, 106.87) mm, rotated rx 180 ry 0 rz 180 deg; joints [-53.163, -15.838, 92.463, 80.169, 54.318, -73.454]
  Call Extruder(5.35652)
  MoveL 6974 to (-36.39, 160.19, 106.87) mm, rotated rx 180 ry 0 rz 180 deg; joints [-53.209, -16.032, 92.605, 80.149, 54.372, -73.401]
  Call Extruder(6.18445)
  MoveL 6975 to (-37.3, 159.15, 106.87) mm, rotated rx 180 ry 0 rz 180 deg; joints [-53.227, -16.229, 92.749, 80.117, 54.398, -73.34]
  Call Extruder(6.35176)
  MoveL 6976 to (-37.47, 158.93, 106.87) mm, rotated rx 180 ry 0 rz -180 deg; joints [-53.227, -16.269, 92.778, 80.109, 54.399, -73.326]
  MoveL 6977 to (-37.47, 158.93, 106.87) mm, rotated rx 180 ry 0 rz -180 deg; joints [-53.227, -16.269, 92.778, 80.109, 54.399, -73.326]
  Call Extruder(6.68519)
  MoveL 6978 to (-37.79, 158.48, 106.87) mm, rotated rx 180 ry 0 rz 180 deg; joints [-53.226, -16.348, 92.835, 80.094, 54.402, -73.299]
  MoveL 6979 to (-37.79, 158.48, 106.87) mm, rotated rx 180 ry 0 rz 180 deg; joints [-53.226, -16.348, 92.835, 80.094, 54.402, -73.299]
  Call Extruder(7.01743)
  MoveL 6980 to (-38.12, 158.03, 106.87) mm, rotated rx 180 ry 0 rz 180 deg; joints [-53.224, -16.428, 92.893, 80.078, 54.405, -73.272]
  MoveL 6981 to (-38.12, 158.03, 106.87) mm, rotated rx 180 ry 0 rz 180 deg; joints [-53.224, -16.428, 92.893, 80.078, 54.405, -73.272]
  Call Extruder(7.13511)
  MoveL 6982 to (-38.22, 157.85, 106.87) mm, rotated rx 180 ry 0 rz 180 deg; joints [-53.221, -16.457, 92.914, 80.071, 54.402, -73.262]
  MoveL 6983 to (-38.22, 157.85, 106.87) mm, rotated rx 180 ry 0 rz 180 deg; joints [-53.221, -16.457, 92.914, 80.071, 54.402, -73.262]
  Call Extruder(7.34283)
  MoveL 6984 to (-38.4, 157.55, 106.87) mm, rotated rx 180 ry 0 rz 180 deg; joints [-53.214, -16.506, 92.95, 80.059, 54.398, -73.244]
  MoveL 6985 to (-38.4, 157.55, 106.87) mm, rotated rx 180 ry 0 rz 180 deg; joints [-53.214, -16.506, 92.95, 80.059, 54.398, -73.244]
  Call Extruder(7.54978)
  MoveL 6986 to (-38.57, 157.25, 106.87) mm, rotated rx 180 ry 0 rz 180 deg; joints [-53.207, -16.556, 92.985, 80.046, 54.394, -73.226]
  MoveL 6987 to (-38.57, 157.25, 106.87) mm, rotated rx 180 ry 0 rz 180 deg; joints [-53.207, -16.556, 92.985, 80.046, 54.394, -73.226]
  Call Extruder(7.75595)
  MoveL 6988 to (-38.75, 156.94, 106.87) mm, rotated rx 180 ry 0 rz 180 deg; joints [-53.2, -16.606, 93.021, 80.034, 54.39, -73.207]
  MoveL 6989 to (-38.75, 156.94, 106.87) mm, rotated rx 180 ry 0 rz 180 deg; joints [-53.2, -16.606, 93.021, 80.034, 54.39, -73.207]
  Call Extruder(7.93763)
  MoveL 6990 to (-38.89, 156.67, 106.87) mm, rotated rx 180 ry 0 rz 180 deg; joints [-53.191, -16.65, 93.053, 80.022, 54.383, -73.191]
  MoveL 6991 to (-38.89, 156.67, 106.87) mm, rotated rx 180 ry 0 rz 180 deg; joints [-53.191, -16.65, 93.053, 80.022, 54.383, -73.191]
  Call Extruder(8.09561)
  MoveL 6992 to (-39, 156.42, 106.87) mm, rotated rx 180 ry 0 rz 180 deg; joints [-53.18, -16.687, 93.08, 80.011, 54.375, -73.176]
  MoveL 6993 to (-39, 156.42, 106.87) mm, rotated rx 180 ry 0 rz 180 deg; joints [-53.18, -16.687, 93.08, 80.011, 54.375, -73.176]
  Call Extruder(8.25300)
  MoveL 6994 to (-39.11, 156.17, 106.87) mm, rotated rx 180 ry 0 rz 180 deg; joints [-53.17, -16.725, 93.107, 80, 54.367, -73.161]
  MoveL 6995 to (-39.11, 156.17, 106.87) mm, rotated rx 180 ry 0 rz 180 deg; joints [-53.17, -16.725, 93.107, 80, 54.367, -73.161]
  Call Extruder(8.43571)
  MoveL 6996 to (-39.23, 155.87, 106.87) mm, rotated rx 180 ry 0 rz 180 deg; joints [-53.156, -16.769, 93.138, 79.986, 54.356, -73.143]
  MoveL 6997 to (-39.23, 155.87, 106.87) mm, rotated rx 180 ry 0 rz 180 deg; joints [-53.156, -16.769, 93.138, 79.986, 54.356, -73.143]
  Call Extruder(8.61768)
  MoveL 6998 to (-39.35, 155.58, 106.87) mm, rotated rx 180 ry 0 rz 180 deg; joints [-53.143, -16.812, 93.17, 79.973, 54.346, -73.125]
  MoveL 6999 to (-39.35, 155.58, 106.87) mm, rotated rx 180 ry 0 rz 180 deg; joints [-53.143, -16.812, 93.17, 79.973, 54.346, -73.125]
  Call Extruder(8.76501)
  MoveL 7000 to (-39.44, 155.34, 106.87) mm, rotated rx 180 ry 0 rz -180 deg; joints [-53.131, -16.848, 93.195, 79.961, 54.336, -73.111]
  MoveL 7001 to (-39.44, 155.34, 106.87) mm, rotated rx 180 ry 0 rz -180 deg; joints [-53.131, -16.848, 93.195, 79.961, 54.336, -73.111]
  Call Extruder(8.87825)
  MoveL 7002 to (-39.5, 155.15, 106.87) mm, rotated rx 180 ry 0 rz 180 deg; joints [-53.121, -16.875, 93.214, 79.952, 54.327, -73.099]
  MoveL 7003 to (-39.5, 155.15, 106.87) mm, rotated rx 180 ry 0 rz 180 deg; joints [-53.121, -16.875, 93.214, 79.952, 54.327, -73.099]
  Call Extruder(8.99104)
  MoveL 7004 to (-39.56, 154.97, 106.87) mm, rotated rx 180 ry 0 rz 180 deg; joints [-53.11, -16.901, 93.233, 79.943, 54.318, -73.088]
  MoveL 7005 to (-39.56, 154.97, 106.87) mm, rotated rx 180 ry 0 rz 180 deg; joints [-53.11, -16.901, 93.233, 79.943, 54.318, -73.088]
  Call Extruder(9.10338)
  MoveL 7006 to (-39.62, 154.78, 106.87) mm, rotated rx -180 ry 0 rz 180 deg; joints [-53.099, -16.928, 93.252, 79.934, 54.309, -73.076]
  MoveL 7007 to (-39.62, 154.78, 106.87) mm, rotated rx -180 ry 0 rz 180 deg; joints [-53.099, -16.928, 93.252, 79.934, 54.309, -73.076]
  Call Extruder(9.21528)
  MoveL 7008 to (-39.68, 154.59, 106.87) mm, rotated rx 180 ry 0 rz 180 deg; joints [-53.088, -16.955, 93.271, 79.924, 54.3, -73.065]
  MoveL 7009 to (-39.68, 154.59, 106.87) mm, rotated rx 180 ry 0 rz 180 deg; joints [-53.088, -16.955, 93.271, 79.924, 54.3, -73.065]
  Call Extruder(9.33668)
  MoveL 7010 to (-39.75, 154.38, 106.87) mm, rotated rx 180 ry 0 rz 180 deg; joints [-53.076, -16.984, 93.292, 79.914, 54.29, -73.052]
  MoveL 7011 to (-39.75, 154.38, 106.87) mm, rotated rx 180 ry 0 rz 180 deg; joints [-53.076, -16.984, 93.292, 79.914, 54.29, -73.052]
  Call Extruder(9.46748)
  MoveL 7012 to (-39.81, 154.16, 106.87) mm, rotated rx -180 ry 0 rz 180 deg; joints [-53.063, -17.015, 93.315, 79.903, 54.279, -73.038]
  MoveL 7013 to (-39.81, 154.16, 106.87) mm, rotated rx -180 ry 0 rz 180 deg; joints [-53.063, -17.015, 93.315, 79.903, 54.279, -73.038]
  Call Extruder(9.59770)
  MoveL 7014 to (-39.88, 153.94, 106.87) mm, rotated rx 180 ry 0 rz 180 deg; joints [-53.049, -17.046, 93.337, 79.892, 54.267, -73.025]
  MoveL 7015 to (-39.88, 153.94, 106.87) mm, rotated rx 180 ry 0 rz 180 deg; joints [-53.049, -17.046, 93.337, 79.892, 54.267, -73.025]
  Call Extruder(9.72737)
  MoveL 7016 to (-39.95, 153.71, 106.87) mm, rotated rx 180 ry 0 rz 180 deg; joints [-53.036, -17.078, 93.359, 79.881, 54.256, -73.011]
  MoveL 7017 to (-39.95, 153.71, 106.87) mm, rotated rx 180 ry 0 rz 180 deg; joints [-53.036, -17.078, 93.359, 79.881, 54.256, -73.011]
  Call Extruder(9.85647)
  MoveL 7018 to (-40.02, 153.49, 106.87) mm, rotated rx 180 ry 0 rz 180 deg; joints [-53.022, -17.109, 93.381, 79.869, 54.245, -72.997]
  MoveL 7019 to (-40.02, 153.49, 106.87) mm, rotated rx 180 ry 0 rz 180 deg; joints [-53.022, -17.109, 93.381, 79.869, 54.245, -72.997]
  Call Extruder(9.97156)
  MoveL 7020 to (-40.06, 153.28, 106.87) mm, rotated rx -180 ry 0 rz -180 deg; joints [-53.007, -17.136, 93.401, 79.858, 54.232, -72.984]
  MoveL 7021 to (-40.06, 153.28, 106.87) mm, rotated rx -180 ry 0 rz -180 deg; joints [-53.007, -17.136, 93.401, 79.858, 54.232, -72.984]
  Call Extruder(10.08619)
  MoveL 7022 to (-40.11, 153.08, 106.87) mm, rotated rx 180 ry 0 rz 180 deg; joints [-52.993, -17.163, 93.42, 79.848, 54.219, -72.972]
  MoveL 7023 to (-40.11, 153.08, 106.87) mm, rotated rx 180 ry 0 rz 180 deg; joints [-52.993, -17.163, 93.42, 79.848, 54.219, -72.972]
  Call Extruder(10.20037)
  MoveL 7024 to (-40.15, 152.88, 106.87) mm, rotated rx 180 ry 0 rz 180 deg; joints [-52.978, -17.19, 93.439, 79.837, 54.207, -72.959]
  MoveL 7025 to (-40.15, 152.88, 106.87) mm, rotated rx 180 ry 0 rz 180 deg; joints [-52.978, -17.19, 93.439, 79.837, 54.207, -72.959]
  Call Extruder(10.31410)
  MoveL 7026 to (-40.2, 152.67, 106.87) mm, rotated rx 180 ry 0 rz 180 deg; joints [-52.963, -17.217, 93.458, 79.826, 54.194, -72.946]
  MoveL 7027 to (-40.2, 152.67, 106.87) mm, rotated rx 180 ry 0 rz 180 deg; joints [-52.963, -17.217, 93.458, 79.826, 54.194, -72.946]
  Call Extruder(10.43953)
  MoveL 7028 to (-40.24, 152.44, 106.87) mm, rotated rx 180 ry 0 rz -180 deg; joints [-52.946, -17.247, 93.479, 79.814, 54.179, -72.932]
  MoveL 7029 to (-40.24, 152.44, 106.87) mm, rotated rx 180 ry 0 rz -180 deg; joints [-52.946, -17.247, 93.479, 79.814, 54.179, -72.932]
  Call Extruder(10.57651)
  MoveL 7030 to (-40.29, 152.2, 106.87) mm, rotated rx 180 ry 0 rz -180 deg; joints [-52.928, -17.28, 93.503, 79.8, 54.163, -72.917]
  MoveL 7031 to (-40.29, 152.2, 106.87) mm, rotated rx 180 ry 0 rz -180 deg; joints [-52.928, -17.28, 93.503, 79.8, 54.163, -72.917]
  Call Extruder(10.71287)
  MoveL 7032 to (-40.34, 151.95, 106.87) mm, rotated rx 180 ry 0 rz 180 deg; joints [-52.909, -17.312, 93.526, 79.786, 54.147, -72.901]
  MoveL 7033 to (-40.34, 151.95, 106.87) mm, rotated rx 180 ry 0 rz 180 deg; joints [-52.909, -17.312, 93.526, 79.786, 54.147, -72.901]
  Call Extruder(10.84863)
  MoveL 7034 to (-40.39, 151.7, 106.87) mm, rotated rx 180 ry 0 rz 180 deg; joints [-52.89, -17.345, 93.549, 79.773, 54.131, -72.886]
  MoveL 7035 to (-40.39, 151.7, 106.87) mm, rotated rx 180 ry 0 rz 180 deg; joints [-52.89, -17.345, 93.549, 79.773, 54.131, -72.886]
  Call Extruder(10.98377)
  MoveL 7036 to (-40.44, 151.45, 106.87) mm, rotated rx -180 ry 0 rz -180 deg; joints [-52.871, -17.377, 93.572, 79.759, 54.114, -72.87]
  MoveL 7037 to (-40.44, 151.45, 106.87) mm, rotated rx -180 ry 0 rz -180 deg; joints [-52.871, -17.377, 93.572, 79.759, 54.114, -72.87]
  Call Extruder(11.11831)
  MoveL 7038 to (-40.49, 151.2, 106.87) mm, rotated rx 180 ry 0 rz 180 deg; joints [-52.853, -17.41, 93.595, 79.746, 54.098, -72.855]
  MoveL 7039 to (-40.49, 151.2, 106.87) mm, rotated rx 180 ry 0 rz 180 deg; joints [-52.853, -17.41, 93.595, 79.746, 54.098, -72.855]
  Call Extruder(11.25223)
  MoveL 7040 to (-40.54, 150.95, 106.87) mm, rotated rx 180 ry 0 rz 180 deg; joints [-52.834, -17.442, 93.618, 79.732, 54.082, -72.839]
  MoveL 7041 to (-40.54, 150.95, 106.87) mm, rotated rx 180 ry 0 rz 180 deg; joints [-52.834, -17.442, 93.618, 79.732, 54.082, -72.839]
  Call Extruder(11.40009)
  MoveL 7042 to (-40.59, 150.67, 106.87) mm, rotated rx -180 ry 0 rz 180 deg; joints [-52.812, -17.478, 93.643, 79.716, 54.063, -72.822]
  MoveL 7043 to (-40.59, 150.67, 106.87) mm, rotated rx -180 ry 0 rz 180 deg; joints [-52.812, -17.478, 93.643, 79.716, 54.063, -72.822]
  Call Extruder(11.56181)
  MoveL 7044 to (-40.64, 150.37, 106.87) mm, rotated rx 180 ry 0 rz 180 deg; joints [-52.787, -17.517, 93.67, 79.699, 54.041, -72.802]
  MoveL 7045 to (-40.64, 150.37, 106.87) mm, rotated rx 180 ry 0 rz 180 deg; joints [-52.787, -17.517, 93.67, 79.699, 54.041, -72.802]
  Call Extruder(11.72281)
  MoveL 7046 to (-40.69, 150.06, 106.87) mm, rotated rx 180 ry 0 rz 180 deg; joints [-52.762, -17.556, 93.698, 79.682, 54.019, -72.783]
  MoveL 7047 to (-40.69, 150.06, 106.87) mm, rotated rx 180 ry 0 rz 180 deg; joints [-52.762, -17.556, 93.698, 79.682, 54.019, -72.783]
  Call Extruder(11.88308)
  MoveL 7048 to (-40.74, 149.76, 106.87) mm, rotated rx -180 ry 0 rz 180 deg; joints [-52.737, -17.595, 93.725, 79.665, 53.998, -72.764]
  MoveL 7049 to (-40.74, 149.76, 106.87) mm, rotated rx -180 ry 0 rz 180 deg; joints [-52.737, -17.595, 93.725, 79.665, 53.998, -72.764]
  Call Extruder(12.04262)
  MoveL 7050 to (-40.78, 149.45, 106.87) mm, rotated rx -180 ry 0 rz 180 deg; joints [-52.712, -17.633, 93.752, 79.647, 53.976, -72.744]
  MoveL 7051 to (-40.78, 149.45, 106.87) mm, rotated rx -180 ry 0 rz 180 deg; joints [-52.712, -17.633, 93.752, 79.647, 53.976, -72.744]
  Call Extruder(12.20143)
  MoveL 7052 to (-40.83, 149.14, 106.87) mm, rotated rx -180 ry 0 rz -180 deg; joints [-52.687, -17.672, 93.779, 79.63, 53.954, -72.725]
  MoveL 7053 to (-40.83, 149.14, 106.87) mm, rotated rx -180 ry 0 rz -180 deg; joints [-52.687, -17.672, 93.779, 79.63, 53.954, -72.725]
  Call Extruder(12.38010)
  MoveL 7054 to (-40.88, 148.8, 106.87) mm, rotated rx 180 ry 0 rz -180 deg; joints [-52.658, -17.715, 93.81, 79.61, 53.928, -72.703]
  MoveL 7055 to (-40.88, 148.8, 106.87) mm, rotated rx 180 ry 0 rz -180 deg; joints [-52.658, -17.715, 93.81, 79.61, 53.928, -72.703]
  Call Extruder(12.57854)
  MoveL 7056 to (-40.93, 148.41, 106.87) mm, rotated rx 180 ry 0 rz 180 deg; joints [-52.624, -17.763, 93.843, 79.587, 53.898, -72.678]
  MoveL 7057 to (-40.93, 148.41, 106.87) mm, rotated rx 180 ry 0 rz 180 deg; joints [-52.624, -17.763, 93.843, 79.587, 53.898, -72.678]
  Call Extruder(12.77611)
  MoveL 7058 to (-40.97, 148.02, 106.87) mm, rotated rx -180 ry 0 rz -180 deg; joints [-52.59, -17.811, 93.876, 79.564, 53.869, -72.653]
  MoveL 7059 to (-40.97, 148.02, 106.87) mm, rotated rx -180 ry 0 rz -180 deg; joints [-52.59, -17.811, 93.876, 79.564, 53.869, -72.653]
  Call Extruder(12.97282)
  MoveL 7060 to (-41.02, 147.63, 106.87) mm, rotated rx -180 ry 0 rz 180 deg; joints [-52.556, -17.859, 93.91, 79.541, 53.839, -72.628]
  MoveL 7061 to (-41.02, 147.63, 106.87) mm, rotated rx -180 ry 0 rz 180 deg; joints [-52.556, -17.859, 93.91, 79.541, 53.839, -72.628]
  Call Extruder(13.16865)
  MoveL 7062 to (-41.06, 147.25, 106.87) mm, rotated rx 180 ry 0 rz -180 deg; joints [-52.521, -17.906, 93.943, 79.518, 53.809, -72.603]
  MoveL 7063 to (-41.06, 147.25, 106.87) mm, rotated rx 180 ry 0 rz -180 deg; joints [-52.521, -17.906, 93.943, 79.518, 53.809, -72.603]
  Call Extruder(13.46405)
  MoveL 7064 to (-41.11, 146.66, 106.87) mm, rotated rx 180 ry 0 rz 180 deg; joints [-52.466, -17.977, 93.992, 79.482, 53.76, -72.565]
  MoveL 7065 to (-41.11, 146.66, 106.87) mm, rotated rx 180 ry 0 rz 180 deg; joints [-52.466, -17.977, 93.992, 79.482, 53.76, -72.565]
  Call Extruder(13.75812)
  MoveL 7066 to (-41.15, 146.07, 106.87) mm, rotated rx 180 ry 0 rz 180 deg; joints [-52.411, -18.047, 94.041, 79.446, 53.711, -72.527]
  MoveL 7067 to (-41.15, 146.07, 106.87) mm, rotated rx 180 ry 0 rz 180 deg; joints [-52.411, -18.047, 94.041, 79.446, 53.711, -72.527]
  Call Extruder(14.05086)
  MoveL 7068 to (-41.2, 145.48, 106.87) mm, rotated rx -180 ry 0 rz 180 deg; joints [-52.355, -18.117, 94.09, 79.41, 53.662, -72.488]
  MoveL 7069 to (-41.2, 145.48, 106.87) mm, rotated rx -180 ry 0 rz 180 deg; joints [-52.355, -18.117, 94.09, 79.41, 53.662, -72.488]
  Call Extruder(14.62431)
  MoveL 7070 to (-41.25, 144.32, 106.87) mm, rotated rx 180 ry 0 rz 180 deg; joints [-52.239, -18.252, 94.183, 79.337, 53.558, -72.412]
  MoveL 7071 to (-41.25, 144.32, 106.87) mm, rotated rx 180 ry 0 rz 180 deg; joints [-52.239, -18.252, 94.183, 79.337, 53.558, -72.412]
  Call Extruder(15.33827)
  MoveL 7072 to (-41.29, 142.86, 106.87) mm, rotated rx -180 ry 0 rz 180 deg; joints [-52.09, -18.418, 94.298, 79.243, 53.426, -72.316]
  Call Extruder(57.40309)
  MoveL 7073 to (-41.29, 57.14, 106.87) mm, rotated rx 180 ry 0 rz 180 deg; joints [-40.759, -27.091, 99.621, 70.797, 43.737, -64.263]
  Call Extruder(57.83165)
  MoveL 7074 to (-41.27, 56.26, 106.87) mm, rotated rx -180 ry 0 rz 180 deg; joints [-40.614, -27.167, 99.662, 70.671, 43.618, -64.149]
  MoveL 7075 to (-41.27, 56.26, 106.87) mm, rotated rx -180 ry 0 rz 180 deg; joints [-40.614, -27.167, 99.662, 70.671, 43.618, -64.149]
  Call Extruder(58.11773)
  MoveL 7076 to (-41.25, 55.68, 106.87) mm, rotated rx 180 ry 0 rz 180 deg; joints [-40.517, -27.216, 99.688, 70.587, 43.538, -64.073]
  MoveL 7077 to (-41.25, 55.68, 106.87) mm, rotated rx 180 ry 0 rz 180 deg; joints [-40.517, -27.216, 99.688, 70.587, 43.538, -64.073]
  Call Extruder(58.69247)
  MoveL 7078 to (-41.2, 54.52, 106.87) mm, rotated rx 180 ry 0 rz 180 deg; joints [-40.32, -27.314, 99.74, 70.416, 43.377, -63.92]
  MoveL 7079 to (-41.2, 54.52, 106.87) mm, rotated rx 180 ry 0 rz 180 deg; joints [-40.32, -27.314, 99.74, 70.416, 43.377, -63.92]
  Call Extruder(58.98587)
  MoveL 7080 to (-41.15, 53.93, 106.87) mm, rotated rx -180 ry 0 rz 180 deg; joints [-40.217, -27.361, 99.765, 70.328, 43.291, -63.842]
  MoveL 7081 to (-41.15, 53.93, 106.87) mm, rotated rx -180 ry 0 rz 180 deg; joints [-40.217, -27.361, 99.765, 70.328, 43.291, -63.842]
  Call Extruder(59.28060)
  MoveL 7082 to (-41.11, 53.34, 106.87) mm, rotated rx 180 ry 0 rz 180 deg; joints [-40.114, -27.408, 99.79, 70.239, 43.206, -63.763]
  MoveL 7083 to (-41.11, 53.34, 106.87) mm, rotated rx 180 ry 0 rz 180 deg; joints [-40.114, -27.408, 99.79, 70.239, 43.206, -63.763]
  Call Extruder(59.57666)
  MoveL 7084 to (-41.06, 52.75, 106.87) mm, rotated rx 180 ry 0 rz 180 deg; joints [-40.01, -27.454, 99.815, 70.15, 43.12, -63.684]
  MoveL 7085 to (-41.06, 52.75, 106.87) mm, rotated rx 180 ry 0 rz 180 deg; joints [-40.01, -27.454, 99.815, 70.15, 43.12, -63.684]
  Call Extruder(59.77293)
  MoveL 7086 to (-41.02, 52.37, 106.87) mm, rotated rx 180 ry 0 rz 180 deg; joints [-39.939, -27.483, 99.831, 70.091, 43.062, -63.632]
  MoveL 7087 to (-41.02, 52.37, 106.87) mm, rotated rx 180 ry 0 rz 180 deg; joints [-39.939, -27.483, 99.831, 70.091, 43.062, -63.632]
  Call Extruder(59.97007)
  MoveL 7088 to (-40.97, 51.98, 106.87) mm, rotated rx 180 ry 0 rz 180 deg; joints [-39.869, -27.512, 99.846, 70.031, 43.003, -63.579]
  MoveL 7089 to (-40.97, 51.98, 106.87) mm, rotated rx 180 ry 0 rz 180 deg; joints [-39.869, -27.512, 99.846, 70.031, 43.003, -63.579]
  Call Extruder(60.16808)
  MoveL 7090 to (-40.92, 51.59, 106.87) mm, rotated rx 180 ry 0 rz 180 deg; joints [-39.798, -27.541, 99.861, 69.971, 42.944, -63.527]
  MoveL 7091 to (-40.92, 51.59, 106.87) mm, rotated rx 180 ry 0 rz 180 deg; joints [-39.798, -27.541, 99.861, 69.971, 42.944, -63.527]
  Call Extruder(60.36695)
  MoveL 7092 to (-40.88, 51.2, 106.87) mm, rotated rx 180 ry 0 rz 180 deg; joints [-39.727, -27.57, 99.876, 69.911, 42.885, -63.474]
  MoveL 7093 to (-40.88, 51.2, 106.87) mm, rotated rx 180 ry 0 rz 180 deg; joints [-39.727, -27.57, 99.876, 69.911, 42.885, -63.474]
  Call Extruder(60.54603)
  MoveL 7094 to (-40.83, 50.86, 106.87) mm, rotated rx -180 ry 0 rz 180 deg; joints [-39.663, -27.595, 99.89, 69.857, 42.832, -63.427]
  MoveL 7095 to (-40.83, 50.86, 106.87) mm, rotated rx -180 ry 0 rz 180 deg; joints [-39.663, -27.595, 99.89, 69.857, 42.832, -63.427]
  Call Extruder(60.70521)
  MoveL 7096 to (-40.78, 50.55, 106.87) mm, rotated rx 180 ry 0 rz 180 deg; joints [-39.605, -27.617, 99.901, 69.808, 42.784, -63.385]
  MoveL 7097 to (-40.78, 50.55, 106.87) mm, rotated rx 180 ry 0 rz 180 deg; joints [-39.605, -27.617, 99.901, 69.808, 42.784, -63.385]
  Call Extruder(60.86512)
  MoveL 7098 to (-40.74, 50.24, 106.87) mm, rotated rx -180 ry 0 rz 180 deg; joints [-39.547, -27.638, 99.912, 69.76, 42.736, -63.343]
  MoveL 7099 to (-40.74, 50.24, 106.87) mm, rotated rx -180 ry 0 rz 180 deg; joints [-39.547, -27.638, 99.912, 69.76, 42.736, -63.343]
  Call Extruder(61.02575)
  MoveL 7100 to (-40.69, 49.94, 106.87) mm, rotated rx 180 ry 0 rz 180 deg; joints [-39.489, -27.659, 99.924, 69.711, 42.688, -63.301]
  MoveL 7101 to (-40.69, 49.94, 106.87) mm, rotated rx 180 ry 0 rz 180 deg; joints [-39.489, -27.659, 99.924, 69.711, 42.688, -63.301]
  Call Extruder(61.18711)
  MoveL 7102 to (-40.64, 49.63, 106.87) mm, rotated rx 180 ry 0 rz 180 deg; joints [-39.431, -27.681, 99.935, 69.663, 42.639, -63.259]
  MoveL 7103 to (-40.64, 49.63, 106.87) mm, rotated rx 180 ry 0 rz 180 deg; joints [-39.431, -27.681, 99.935, 69.663, 42.639, -63.259]
  Call Extruder(61.34920)
  MoveL 7104 to (-40.59, 49.33, 106.87) mm, rotated rx 180 ry 0 rz 180 deg; joints [-39.373, -27.702, 99.946, 69.614, 42.591, -63.216]
  MoveL 7105 to (-40.59, 49.33, 106.87) mm, rotated rx 180 ry 0 rz 180 deg; joints [-39.373, -27.702, 99.946, 69.614, 42.591, -63.216]
  Call Extruder(61.49740)
  MoveL 7106 to (-40.54, 49.05, 106.87) mm, rotated rx 180 ry 0 rz 180 deg; joints [-39.32, -27.721, 99.956, 69.569, 42.546, -63.178]
  MoveL 7107 to (-40.54, 49.05, 106.87) mm, rotated rx 180 ry 0 rz 180 deg; joints [-39.32, -27.721, 99.956, 69.569, 42.546, -63.178]
  Call Extruder(61.63163)
  MoveL 7108 to (-40.49, 48.8, 106.87) mm, rotated rx -180 ry 0 rz 180 deg; joints [-39.271, -27.737, 99.964, 69.529, 42.506, -63.143]
  MoveL 7109 to (-40.49, 48.8, 106.87) mm, rotated rx -180 ry 0 rz 180 deg; joints [-39.271, -27.737, 99.964, 69.529, 42.506, -63.143]
  Call Extruder(61.76647)
  MoveL 7110 to (-40.44, 48.55, 106.87) mm, rotated rx 180 ry 0 rz 180 deg; joints [-39.222, -27.753, 99.973, 69.488, 42.465, -63.108]
  MoveL 7111 to (-40.44, 48.55, 106.87) mm, rotated rx 180 ry 0 rz 180 deg; joints [-39.222, -27.753, 99.973, 69.488, 42.465, -63.108]
  Call Extruder(61.90192)
  MoveL 7112 to (-40.39, 48.3, 106.87) mm, rotated rx 180 ry 0 rz 180 deg; joints [-39.174, -27.769, 99.981, 69.448, 42.424, -63.074]
  MoveL 7113 to (-40.39, 48.3, 106.87) mm, rotated rx 180 ry 0 rz 180 deg; joints [-39.174, -27.769, 99.981, 69.448, 42.424, -63.074]
  Call Extruder(62.03798)
  MoveL 7114 to (-40.34, 48.05, 106.87) mm, rotated rx -180 ry 0 rz 180 deg; joints [-39.125, -27.785, 99.99, 69.407, 42.383, -63.039]
  MoveL 7115 to (-40.34, 48.05, 106.87) mm, rotated rx -180 ry 0 rz 180 deg; joints [-39.125, -27.785, 99.99, 69.407, 42.383, -63.039]
  Call Extruder(62.17465)
  MoveL 7116 to (-40.29, 47.8, 106.87) mm, rotated rx 180 ry 0 rz 180 deg; joints [-39.076, -27.801, 99.998, 69.366, 42.342, -63.004]
  MoveL 7117 to (-40.29, 47.8, 106.87) mm, rotated rx 180 ry 0 rz 180 deg; joints [-39.076, -27.801, 99.998, 69.366, 42.342, -63.004]
  Call Extruder(62.31193)
  MoveL 7118 to (-40.24, 47.55, 106.87) mm, rotated rx 180 ry 0 rz 180 deg; joints [-39.027, -27.817, 100.007, 69.325, 42.301, -62.969]
  MoveL 7119 to (-40.24, 47.55, 106.87) mm, rotated rx 180 ry 0 rz 180 deg; joints [-39.027, -27.817, 100.007, 69.325, 42.301, -62.969]
  Call Extruder(62.43760)
  MoveL 7120 to (-40.2, 47.33, 106.87) mm, rotated rx 180 ry 0 rz 180 deg; joints [-38.982, -27.832, 100.014, 69.288, 42.264, -62.937]
  MoveL 7121 to (-40.2, 47.33, 106.87) mm, rotated rx 180 ry 0 rz 180 deg; joints [-38.982, -27.832, 100.014, 69.288, 42.264, -62.937]
  Call Extruder(62.55156)
  MoveL 7122 to (-40.15, 47.12, 106.87) mm, rotated rx 180 ry 0 rz 180 deg; joints [-38.941, -27.845, 100.021, 69.254, 42.229, -62.908]
  MoveL 7123 to (-40.15, 47.12, 106.87) mm, rotated rx 180 ry 0 rz 180 deg; joints [-38.941, -27.845, 100.021, 69.254, 42.229, -62.908]
  Call Extruder(62.66597)
  MoveL 7124 to (-40.11, 46.92, 106.87) mm, rotated rx 180 ry 0 rz 180 deg; joints [-38.9, -27.857, 100.028, 69.22, 42.195, -62.879]
  MoveL 7125 to (-40.11, 46.92, 106.87) mm, rotated rx 180 ry 0 rz 180 deg; joints [-38.9, -27.857, 100.028, 69.22, 42.195, -62.879]
  Call Extruder(62.78083)
  MoveL 7126 to (-40.06, 46.72, 106.87) mm, rotated rx 180 ry 0 rz 180 deg; joints [-38.859, -27.87, 100.034, 69.186, 42.161, -62.85]
  MoveL 7127 to (-40.06, 46.72, 106.87) mm, rotated rx 180 ry 0 rz 180 deg; joints [-38.859, -27.87, 100.034, 69.186, 42.161, -62.85]
  Call Extruder(62.89614)
  MoveL 7128 to (-40.02, 46.51, 106.87) mm, rotated rx 180 ry 0 rz 180 deg; joints [-38.819, -27.882, 100.041, 69.152, 42.127, -62.821]
  MoveL 7129 to (-40.02, 46.51, 106.87) mm, rotated rx 180 ry 0 rz 180 deg; joints [-38.819, -27.882, 100.041, 69.152, 42.127, -62.821]
  Call Extruder(63.02552)
  MoveL 7130 to (-39.95, 46.29, 106.87) mm, rotated rx -180 ry 0 rz 180 deg; joints [-38.771, -27.894, 100.047, 69.114, 42.087, -62.789]
  MoveL 7131 to (-39.95, 46.29, 106.87) mm, rotated rx -180 ry 0 rz 180 deg; joints [-38.771, -27.894, 100.047, 69.114, 42.087, -62.789]
  Call Extruder(63.15547)
  MoveL 7132 to (-39.88, 46.06, 106.87) mm, rotated rx 180 ry 0 rz 180 deg; joints [-38.724, -27.906, 100.053, 69.076, 42.046, -62.757]
  MoveL 7133 to (-39.88, 46.06, 106.87) mm, rotated rx 180 ry 0 rz 180 deg; joints [-38.724, -27.906, 100.053, 69.076, 42.046, -62.757]
  Call Extruder(63.28598)
  MoveL 7134 to (-39.81, 45.84, 106.87) mm, rotated rx 180 ry 0 rz 180 deg; joints [-38.677, -27.918, 100.059, 69.038, 42.007, -62.725]
  MoveL 7135 to (-39.81, 45.84, 106.87) mm, rotated rx 180 ry 0 rz 180 deg; joints [-38.677, -27.918, 100.059, 69.038, 42.007, -62.725]
  Call Extruder(63.41705)
  MoveL 7136 to (-39.75, 45.62, 106.87) mm, rotated rx -180 ry 0 rz 180 deg; joints [-38.629, -27.93, 100.065, 68.999, 41.966, -62.693]
  MoveL 7137 to (-39.75, 45.62, 106.87) mm, rotated rx -180 ry 0 rz 180 deg; joints [-38.629, -27.93, 100.065, 68.999, 41.966, -62.693]
  Call Extruder(63.53870)
  MoveL 7138 to (-39.68, 45.41, 106.87) mm, rotated rx 180 ry 0 rz 180 deg; joints [-38.585, -27.94, 100.071, 68.964, 41.929, -62.664]
  MoveL 7139 to (-39.68, 45.41, 106.87) mm, rotated rx 180 ry 0 rz 180 deg; joints [-38.585, -27.94, 100.071, 68.964, 41.929, -62.664]
  Call Extruder(63.65082)
  MoveL 7140 to (-39.62, 45.22, 106.87) mm, rotated rx 180 ry 0 rz -180 deg; joints [-38.544, -27.95, 100.076, 68.931, 41.895, -62.637]
  MoveL 7141 to (-39.62, 45.22, 106.87) mm, rotated rx 180 ry 0 rz -180 deg; joints [-38.544, -27.95, 100.076, 68.931, 41.895, -62.637]
  Call Extruder(63.76339)
  MoveL 7142 to (-39.56, 45.03, 106.87) mm, rotated rx 180 ry 0 rz 180 deg; joints [-38.504, -27.959, 100.081, 68.898, 41.86, -62.61]
  MoveL 7143 to (-39.56, 45.03, 106.87) mm, rotated rx 180 ry 0 rz 180 deg; joints [-38.504, -27.959, 100.081, 68.898, 41.86, -62.61]
  Call Extruder(63.87640)
  MoveL 7144 to (-39.5, 44.85, 106.87) mm, rotated rx 180 ry 0 rz 180 deg; joints [-38.463, -27.969, 100.086, 68.866, 41.826, -62.582]
  MoveL 7145 to (-39.5, 44.85, 106.87) mm, rotated rx 180 ry 0 rz 180 deg; joints [-38.463, -27.969, 100.086, 68.866, 41.826, -62.582]
  Call Extruder(63.98986)
  MoveL 7146 to (-39.44, 44.66, 106.87) mm, rotated rx -180 ry 0 rz 180 deg; joints [-38.422, -27.978, 100.091, 68.833, 41.791, -62.555]
  MoveL 7147 to (-39.44, 44.66, 106.87) mm, rotated rx -180 ry 0 rz 180 deg; joints [-38.422, -27.978, 100.091, 68.833, 41.791, -62.555]
  Call Extruder(64.13750)
  MoveL 7148 to (-39.35, 44.42, 106.87) mm, rotated rx 180 ry 0 rz 180 deg; joints [-38.369, -27.989, 100.096, 68.791, 41.745, -62.52]
  MoveL 7149 to (-39.35, 44.42, 106.87) mm, rotated rx 180 ry 0 rz 180 deg; joints [-38.369, -27.989, 100.096, 68.791, 41.745, -62.52]
  Call Extruder(64.31984)
  MoveL 7150 to (-39.23, 44.12, 106.87) mm, rotated rx 180 ry 0 rz 180 deg; joints [-38.302, -28, 100.102, 68.738, 41.688, -62.478]
  MoveL 7151 to (-39.23, 44.12, 106.87) mm, rotated rx 180 ry 0 rz 180 deg; joints [-38.302, -28, 100.102, 68.738, 41.688, -62.478]
  Call Extruder(64.50294)
  MoveL 7152 to (-39.11, 43.83, 106.87) mm, rotated rx -180 ry 0 rz 180 deg; joints [-38.236, -28.012, 100.108, 68.686, 41.631, -62.436]
  MoveL 7153 to (-39.11, 43.83, 106.87) mm, rotated rx -180 ry 0 rz 180 deg; joints [-38.236, -28.012, 100.108, 68.686, 41.631, -62.436]
  Call Extruder(64.66062)
  MoveL 7154 to (-39, 43.58, 106.87) mm, rotated rx 180 ry 0 rz -180 deg; joints [-38.178, -28.021, 100.113, 68.641, 41.582, -62.399]
  MoveL 7155 to (-39, 43.58, 106.87) mm, rotated rx 180 ry 0 rz -180 deg; joints [-38.178, -28.021, 100.113, 68.641, 41.582, -62.399]
  Call Extruder(64.81891)
  MoveL 7156 to (-38.89, 43.34, 106.87) mm, rotated rx 180 ry 0 rz 180 deg; joints [-38.121, -28.031, 100.118, 68.597, 41.533, -62.363]
  MoveL 7157 to (-38.89, 43.34, 106.87) mm, rotated rx 180 ry 0 rz 180 deg; joints [-38.121, -28.031, 100.118, 68.597, 41.533, -62.363]
  Call Extruder(65.00093)
  MoveL 7158 to (-38.75, 43.06, 106.87) mm, rotated rx 180 ry 0 rz 180 deg; joints [-38.054, -28.039, 100.122, 68.546, 41.475, -62.322]
  MoveL 7159 to (-38.75, 43.06, 106.87) mm, rotated rx 180 ry 0 rz 180 deg; joints [-38.054, -28.039, 100.122, 68.546, 41.475, -62.322]
  Call Extruder(65.20748)
  MoveL 7160 to (-38.57, 42.75, 106.87) mm, rotated rx 180 ry 0 rz 180 deg; joints [-37.977, -28.046, 100.126, 68.489, 41.408, -62.278]
  MoveL 7161 to (-38.57, 42.75, 106.87) mm, rotated rx 180 ry 0 rz 180 deg; joints [-37.977, -28.046, 100.126, 68.489, 41.408, -62.278]
  Call Extruder(65.41482)
  MoveL 7162 to (-38.4, 42.45, 106.87) mm, rotated rx 180 ry 0 rz 180 deg; joints [-37.901, -28.052, 100.129, 68.432, 41.342, -62.233]
  MoveL 7163 to (-38.4, 42.45, 106.87) mm, rotated rx 180 ry 0 rz 180 deg; joints [-37.901, -28.052, 100.129, 68.432, 41.342, -62.233]
  Call Extruder(65.62293)
  MoveL 7164 to (-38.22, 42.15, 106.87) mm, rotated rx 180 ry 0 rz 180 deg; joints [-37.825, -28.059, 100.133, 68.374, 41.276, -62.188]
  MoveL 7165 to (-38.22, 42.15, 106.87) mm, rotated rx 180 ry 0 rz 180 deg; joints [-37.825, -28.059, 100.133, 68.374, 41.276, -62.188]
  Call Extruder(65.74065)
  MoveL 7166 to (-38.12, 41.97, 106.87) mm, rotated rx 180 ry 0 rz 180 deg; joints [-37.782, -28.062, 100.134, 68.342, 41.238, -62.163]
  MoveL 7167 to (-38.12, 41.97, 106.87) mm, rotated rx 180 ry 0 rz 180 deg; joints [-37.782, -28.062, 100.134, 68.342, 41.238, -62.163]
  Call Extruder(66.07349)
  MoveL 7168 to (-37.8, 41.52, 106.87) mm, rotated rx 180 ry 0 rz 180 deg; joints [-37.659, -28.064, 100.136, 68.254, 41.13, -62.096]
  MoveL 7169 to (-37.8, 41.52, 106.87) mm, rotated rx 180 ry 0 rz 180 deg; joints [-37.659, -28.064, 100.136, 68.254, 41.13, -62.096]
  Call Extruder(66.40752)
  MoveL 7170 to (-37.47, 41.07, 106.87) mm, rotated rx 180 ry 0 rz 180 deg; joints [-37.537, -28.066, 100.137, 68.165, 41.022, -62.028]
  MoveL 7171 to (-37.47, 41.07, 106.87) mm, rotated rx 180 ry 0 rz 180 deg; joints [-37.537, -28.066, 100.137, 68.165, 41.022, -62.028]
  Call Extruder(66.57511)
  MoveL 7172 to (-37.3, 40.85, 106.87) mm, rotated rx 180 ry 0 rz 180 deg; joints [-37.475, -28.067, 100.137, 68.121, 40.968, -61.995]
  Call Extruder(67.40442)
  MoveL 7173 to (-36.39, 39.81, 106.87) mm, rotated rx -180 ry 0 rz 180 deg; joints [-37.173, -28.054, 100.13, 67.91, 40.699, -61.839]
  Call Extruder(68.03549)
  MoveL 7174 to (-35.61, 39.11, 106.87) mm, rotated rx 180 ry 0 rz 180 deg; joints [-36.947, -28.026, 100.116, 67.76, 40.495, -61.733]
  MoveL 7175 to (-35.61, 39.11, 106.87) mm, rotated rx 180 ry 0 rz 180 deg; joints [-36.947, -28.026, 100.116, 67.76, 40.495, -61.733]
  Call Extruder(68.23306)
  MoveL 7176 to (-35.35, 38.9, 106.87) mm, rotated rx 180 ry 0 rz 180 deg; joints [-36.876, -28.017, 100.111, 67.714, 40.431, -61.701]
  Call Extruder(68.56708)
  MoveL 7177 to (-34.9, 38.57, 106.87) mm, rotated rx -180 ry 0 rz 180 deg; joints [-36.759, -27.994, 100.099, 67.64, 40.324, -61.651]
  MoveL 7178 to (-34.9, 38.57, 106.87) mm, rotated rx -180 ry 0 rz 180 deg; joints [-36.759, -27.994, 100.099, 67.64, 40.324, -61.651]
  Call Extruder(68.89991)
  MoveL 7179 to (-34.45, 38.24, 106.87) mm, rotated rx -180 ry 0 rz -180 deg; joints [-36.642, -27.972, 100.087, 67.566, 40.217, -61.601]
  MoveL 7180 to (-34.45, 38.24, 106.87) mm, rotated rx -180 ry 0 rz -180 deg; joints [-36.642, -27.972, 100.087, 67.566, 40.217, -61.601]
  Call Extruder(69.07916)
  MoveL 7181 to (-34.21, 38.07, 106.87) mm, rotated rx 180 ry 0 rz 180 deg; joints [-36.579, -27.959, 100.081, 67.526, 40.159, -61.574]
  MoveL 7182 to (-34.21, 38.07, 106.87) mm, rotated rx 180 ry 0 rz 180 deg; joints [-36.579, -27.959, 100.081, 67.526, 40.159, -61.574]
  Call Extruder(69.28727)
  MoveL 7183 to (-33.9, 37.89, 106.87) mm, rotated rx 180 ry 0 rz 180 deg; joints [-36.509, -27.941, 100.071, 67.484, 40.094, -61.547]
  MoveL 7184 to (-33.9, 37.89, 106.87) mm, rotated rx 180 ry 0 rz 180 deg; joints [-36.509, -27.941, 100.071, 67.484, 40.094, -61.547]
  Call Extruder(69.49460)
  MoveL 7185 to (-33.6, 37.71, 106.87) mm, rotated rx -180 ry 0 rz 180 deg; joints [-36.439, -27.921, 100.061, 67.442, 40.029, -61.52]
  MoveL 7186 to (-33.6, 37.71, 106.87) mm, rotated rx -180 ry 0 rz 180 deg; joints [-36.439, -27.921, 100.061, 67.442, 40.029, -61.52]
  Call Extruder(69.70115)
  MoveL 7187 to (-33.29, 37.54, 106.87) mm, rotated rx 180 ry 0 rz 180 deg; joints [-36.368, -27.902, 100.051, 67.399, 39.963, -61.493]
  MoveL 7188 to (-33.29, 37.54, 106.87) mm, rotated rx 180 ry 0 rz 180 deg; joints [-36.368, -27.902, 100.051, 67.399, 39.963, -61.493]
  Call Extruder(69.90692)
  MoveL 7189 to (-32.99, 37.36, 106.87) mm, rotated rx 180 ry 0 rz 180 deg; joints [-36.298, -27.883, 100.041, 67.357, 39.898, -61.466]
  MoveL 7190 to (-32.99, 37.36, 106.87) mm, rotated rx 180 ry 0 rz 180 deg; joints [-36.298, -27.883, 100.041, 67.357, 39.898, -61.466]
  Call Extruder(70.06523)
  MoveL 7191 to (-32.74, 37.26, 106.87) mm, rotated rx 180 ry 0 rz 180 deg; joints [-36.247, -27.865, 100.031, 67.329, 39.85, -61.45]
  MoveL 7192 to (-32.74, 37.26, 106.87) mm, rotated rx 180 ry 0 rz 180 deg; joints [-36.247, -27.865, 100.031, 67.329, 39.85, -61.45]
  Call Extruder(70.22293)
  MoveL 7193 to (-32.49, 37.15, 106.87) mm, rotated rx 180 ry 0 rz 180 deg; joints [-36.196, -27.846, 100.022, 67.301, 39.802, -61.433]
  MoveL 7194 to (-32.49, 37.15, 106.87) mm, rotated rx 180 ry 0 rz 180 deg; joints [-36.196, -27.846, 100.022, 67.301, 39.802, -61.433]
  Call Extruder(70.39301)
  MoveL 7195 to (-32.22, 37.04, 106.87) mm, rotated rx -180 ry 0 rz 180 deg; joints [-36.141, -27.826, 100.011, 67.27, 39.75, -61.416]
  MoveL 7196 to (-32.22, 37.04, 106.87) mm, rotated rx -180 ry 0 rz 180 deg; joints [-36.141, -27.826, 100.011, 67.27, 39.75, -61.416]
  Call Extruder(70.57535)
  MoveL 7197 to (-31.93, 36.91, 106.87) mm, rotated rx 180 ry 0 rz 180 deg; joints [-36.082, -27.803, 99.999, 67.238, 39.694, -61.397]
  MoveL 7198 to (-31.93, 36.91, 106.87) mm, rotated rx 180 ry 0 rz 180 deg; joints [-36.082, -27.803, 99.999, 67.238, 39.694, -61.397]
  Call Extruder(70.75692)
  MoveL 7199 to (-31.64, 36.79, 106.87) mm, rotated rx 180 ry 0 rz 180 deg; joints [-36.023, -27.781, 99.987, 67.206, 39.638, -61.378]
  MoveL 7200 to (-31.64, 36.79, 106.87) mm, rotated rx 180 ry 0 rz 180 deg; joints [-36.023, -27.781, 99.987, 67.206, 39.638, -61.378]
  Call Extruder(70.87038)
  MoveL 7201 to (-31.45, 36.73, 106.87) mm, rotated rx 180 ry 0 rz 180 deg; joints [-35.989, -27.765, 99.979, 67.188, 39.605, -61.369]
  MoveL 7202 to (-31.45, 36.73, 106.87) mm, rotated rx 180 ry 0 rz 180 deg; joints [-35.989, -27.765, 99.979, 67.188, 39.605, -61.369]
  Call Extruder(70.98339)
  MoveL 7203 to (-31.26, 36.67, 106.87) mm, rotated rx 180 ry 0 rz 180 deg; joints [-35.954, -27.749, 99.971, 67.17, 39.571, -61.36]
  MoveL 7204 to (-31.26, 36.67, 106.87) mm, rotated rx 180 ry 0 rz 180 deg; joints [-35.954, -27.749, 99.971, 67.17, 39.571, -61.36]
  Call Extruder(71.09596)
  MoveL 7205 to (-31.07, 36.61, 106.87) mm, rotated rx 180 ry 0 rz 180 deg; joints [-35.919, -27.733, 99.963, 67.152, 39.538, -61.35]
  MoveL 7206 to (-31.07, 36.61, 106.87) mm, rotated rx 180 ry 0 rz 180 deg; joints [-35.919, -27.733, 99.963, 67.152, 39.538, -61.35]
  Call Extruder(71.20809)
  MoveL 7207 to (-30.88, 36.55, 106.87) mm, rotated rx -180 ry 0 rz 180 deg; joints [-35.884, -27.718, 99.954, 67.134, 39.504, -61.341]
  MoveL 7208 to (-30.88, 36.55, 106.87) mm, rotated rx -180 ry 0 rz 180 deg; joints [-35.884, -27.718, 99.954, 67.134, 39.504, -61.341]
  Call Extruder(71.31977)
  MoveL 7209 to (-30.7, 36.49, 106.87) mm, rotated rx 180 ry 0 rz 180 deg; joints [-35.849, -27.702, 99.946, 67.117, 39.471, -61.332]
  MoveL 7210 to (-30.7, 36.49, 106.87) mm, rotated rx 180 ry 0 rz 180 deg; joints [-35.849, -27.702, 99.946, 67.117, 39.471, -61.332]
  Call Extruder(71.45084)
  MoveL 7211 to (-30.47, 36.42, 106.87) mm, rotated rx 180 ry 0 rz 180 deg; joints [-35.809, -27.682, 99.936, 67.096, 39.432, -61.321]
  MoveL 7212 to (-30.47, 36.42, 106.87) mm, rotated rx 180 ry 0 rz 180 deg; joints [-35.809, -27.682, 99.936, 67.096, 39.432, -61.321]
  Call Extruder(71.58135)
  MoveL 7213 to (-30.25, 36.35, 106.87) mm, rotated rx 180 ry 0 rz 180 deg; joints [-35.768, -27.663, 99.926, 67.076, 39.393, -61.311]
  MoveL 7214 to (-30.25, 36.35, 106.87) mm, rotated rx 180 ry 0 rz 180 deg; joints [-35.768, -27.663, 99.926, 67.076, 39.393, -61.311]
  Call Extruder(71.71129)
  MoveL 7215 to (-30.02, 36.28, 106.87) mm, rotated rx 180 ry 0 rz 180 deg; joints [-35.728, -27.644, 99.915, 67.056, 39.354, -61.301]
  MoveL 7216 to (-30.02, 36.28, 106.87) mm, rotated rx 180 ry 0 rz 180 deg; joints [-35.728, -27.644, 99.915, 67.056, 39.354, -61.301]
  Call Extruder(71.84067)
  MoveL 7217 to (-29.8, 36.22, 106.87) mm, rotated rx -180 ry 0 rz 180 deg; joints [-35.688, -27.625, 99.905, 67.035, 39.315, -61.29]
  MoveL 7218 to (-29.8, 36.22, 106.87) mm, rotated rx -180 ry 0 rz 180 deg; joints [-35.688, -27.625, 99.905, 67.035, 39.315, -61.29]
  Call Extruder(71.96263)
  MoveL 7219 to (-29.59, 36.16, 106.87) mm, rotated rx 180 ry 0 rz -180 deg; joints [-35.651, -27.605, 99.895, 67.018, 39.279, -61.282]
  MoveL 7220 to (-29.59, 36.16, 106.87) mm, rotated rx 180 ry 0 rz -180 deg; joints [-35.651, -27.605, 99.895, 67.018, 39.279, -61.282]
  Call Extruder(72.07748)
  MoveL 7221 to (-29.38, 36.12, 106.87) mm, rotated rx 180 ry 0 rz 180 deg; joints [-35.617, -27.586, 99.885, 67.002, 39.246, -61.275]
  MoveL 7222 to (-29.38, 36.12, 106.87) mm, rotated rx 180 ry 0 rz 180 deg; joints [-35.617, -27.586, 99.885, 67.002, 39.246, -61.275]
  Call Extruder(72.19188)
  MoveL 7223 to (-29.18, 36.07, 106.87) mm, rotated rx 180 ry 0 rz 180 deg; joints [-35.584, -27.567, 99.875, 66.987, 39.213, -61.268]
  MoveL 7224 to (-29.18, 36.07, 106.87) mm, rotated rx 180 ry 0 rz 180 deg; joints [-35.584, -27.567, 99.875, 66.987, 39.213, -61.268]
  Call Extruder(72.30582)
  MoveL 7225 to (-28.97, 36.03, 106.87) mm, rotated rx 180 ry 0 rz 180 deg; joints [-35.55, -27.549, 99.865, 66.971, 39.18, -61.261]
  MoveL 7226 to (-28.97, 36.03, 106.87) mm, rotated rx 180 ry 0 rz 180 deg; joints [-35.55, -27.549, 99.865, 66.971, 39.18, -61.261]
  Call Extruder(72.41931)
  MoveL 7227 to (-28.77, 35.98, 106.87) mm, rotated rx 180 ry 0 rz 180 deg; joints [-35.517, -27.529, 99.855, 66.956, 39.147, -61.255]
  MoveL 7228 to (-28.77, 35.98, 106.87) mm, rotated rx 180 ry 0 rz 180 deg; joints [-35.517, -27.529, 99.855, 66.956, 39.147, -61.255]
  Call Extruder(72.55659)
  MoveL 7229 to (-28.52, 35.93, 106.87) mm, rotated rx -180 ry 0 rz 180 deg; joints [-35.477, -27.506, 99.842, 66.938, 39.108, -61.247]
  MoveL 7230 to (-28.52, 35.93, 106.87) mm, rotated rx -180 ry 0 rz 180 deg; joints [-35.477, -27.506, 99.842, 66.938, 39.108, -61.247]
  Call Extruder(72.69326)
  MoveL 7231 to (-28.27, 35.88, 106.87) mm, rotated rx 180 ry 0 rz 180 deg; joints [-35.437, -27.482, 99.83, 66.92, 39.068, -61.24]
  MoveL 7232 to (-28.27, 35.88, 106.87) mm, rotated rx 180 ry 0 rz 180 deg; joints [-35.437, -27.482, 99.83, 66.92, 39.068, -61.24]
  Call Extruder(72.82933)
  MoveL 7233 to (-28.02, 35.83, 106.87) mm, rotated rx 180 ry 0 rz 180 deg; joints [-35.397, -27.458, 99.817, 66.902, 39.029, -61.232]
  MoveL 7234 to (-28.02, 35.83, 106.87) mm, rotated rx 180 ry 0 rz 180 deg; joints [-35.397, -27.458, 99.817, 66.902, 39.029, -61.232]
  Call Extruder(72.96478)
  MoveL 7235 to (-27.77, 35.78, 106.87) mm, rotated rx 180 ry 0 rz 180 deg; joints [-35.357, -27.435, 99.805, 66.884, 38.99, -61.225]
  MoveL 7236 to (-27.77, 35.78, 106.87) mm, rotated rx 180 ry 0 rz 180 deg; joints [-35.357, -27.435, 99.805, 66.884, 38.99, -61.225]
  Call Extruder(73.09962)
  MoveL 7237 to (-27.52, 35.73, 106.87) mm, rotated rx 180 ry 0 rz 180 deg; joints [-35.317, -27.411, 99.792, 66.867, 38.951, -61.218]
  MoveL 7238 to (-27.52, 35.73, 106.87) mm, rotated rx 180 ry 0 rz 180 deg; joints [-35.317, -27.411, 99.792, 66.867, 38.951, -61.218]
  Call Extruder(73.23385)
  MoveL 7239 to (-27.28, 35.68, 106.87) mm, rotated rx -180 ry 0 rz 180 deg; joints [-35.277, -27.387, 99.779, 66.849, 38.911, -61.21]
  MoveL 7240 to (-27.28, 35.68, 106.87) mm, rotated rx -180 ry 0 rz 180 deg; joints [-35.277, -27.387, 99.779, 66.849, 38.911, -61.21]
  Call Extruder(73.36747)
  MoveL 7241 to (-27.03, 35.63, 106.87) mm, rotated rx -180 ry 0 rz 180 deg; joints [-35.238, -27.364, 99.767, 66.831, 38.872, -61.203]
  MoveL 7242 to (-27.03, 35.63, 106.87) mm, rotated rx -180 ry 0 rz 180 deg; joints [-35.238, -27.364, 99.767, 66.831, 38.872, -61.203]
  Call Extruder(73.52957)
  MoveL 7243 to (-26.72, 35.59, 106.87) mm, rotated rx -180 ry 0 rz 180 deg; joints [-35.191, -27.333, 99.751, 66.811, 38.826, -61.196]
  MoveL 7244 to (-26.72, 35.59, 106.87) mm, rotated rx -180 ry 0 rz 180 deg; joints [-35.191, -27.333, 99.751, 66.811, 38.826, -61.196]
  Call Extruder(73.69094)
  MoveL 7245 to (-26.41, 35.54, 106.87) mm, rotated rx 180 ry 0 rz 180 deg; joints [-35.145, -27.303, 99.735, 66.792, 38.78, -61.188]
  MoveL 7246 to (-26.41, 35.54, 106.87) mm, rotated rx 180 ry 0 rz 180 deg; joints [-35.145, -27.303, 99.735, 66.792, 38.78, -61.188]
  Call Extruder(73.85158)
  MoveL 7247 to (-26.11, 35.49, 106.87) mm, rotated rx 180 ry 0 rz 180 deg; joints [-35.098, -27.273, 99.718, 66.772, 38.734, -61.181]
  MoveL 7248 to (-26.11, 35.49, 106.87) mm, rotated rx 180 ry 0 rz 180 deg; joints [-35.098, -27.273, 99.718, 66.772, 38.734, -61.181]
  Call Extruder(74.01150)
  MoveL 7249 to (-25.8, 35.44, 106.87) mm, rotated rx 180 ry 0 rz 180 deg; joints [-35.052, -27.243, 99.702, 66.753, 38.688, -61.174]
  MoveL 7250 to (-25.8, 35.44, 106.87) mm, rotated rx 180 ry 0 rz 180 deg; joints [-35.052, -27.243, 99.702, 66.753, 38.688, -61.174]
  Call Extruder(74.17069)
  MoveL 7251 to (-25.5, 35.39, 106.87) mm, rotated rx 180 ry 0 rz 180 deg; joints [-35.006, -27.212, 99.686, 66.733, 38.641, -61.167]
  MoveL 7252 to (-25.5, 35.39, 106.87) mm, rotated rx 180 ry 0 rz 180 deg; joints [-35.006, -27.212, 99.686, 66.733, 38.641, -61.167]
  Call Extruder(74.32915)
  MoveL 7253 to (-25.19, 35.34, 106.87) mm, rotated rx 180 ry 0 rz 180 deg; joints [-34.96, -27.182, 99.67, 66.714, 38.596, -61.16]
  MoveL 7254 to (-25.19, 35.34, 106.87) mm, rotated rx 180 ry 0 rz 180 deg; joints [-34.96, -27.182, 99.67, 66.714, 38.596, -61.16]
  Call Extruder(74.52802)
  MoveL 7255 to (-24.8, 35.3, 106.87) mm, rotated rx 180 ry 0 rz 180 deg; joints [-34.904, -27.143, 99.649, 66.692, 38.54, -61.153]
  MoveL 7256 to (-24.8, 35.3, 106.87) mm, rotated rx 180 ry 0 rz 180 deg; joints [-34.904, -27.143, 99.649, 66.692, 38.54, -61.153]
  Call Extruder(74.72603)
  MoveL 7257 to (-24.42, 35.25, 106.87) mm, rotated rx 180 ry 0 rz 180 deg; joints [-34.849, -27.103, 99.627, 66.67, 38.484, -61.147]
  MoveL 7258 to (-24.42, 35.25, 106.87) mm, rotated rx 180 ry 0 rz 180 deg; joints [-34.849, -27.103, 99.627, 66.67, 38.484, -61.147]
  Call Extruder(74.92317)
  MoveL 7259 to (-24.03, 35.21, 106.87) mm, rotated rx 180 ry 0 rz 180 deg; joints [-34.794, -27.063, 99.606, 66.649, 38.428, -61.14]
  MoveL 7260 to (-24.03, 35.21, 106.87) mm, rotated rx 180 ry 0 rz 180 deg; joints [-34.794, -27.063, 99.606, 66.649, 38.428, -61.14]
  Call Extruder(75.11944)
  MoveL 7261 to (-23.64, 35.16, 106.87) mm, rotated rx 180 ry 0 rz 180 deg; joints [-34.738, -27.023, 99.585, 66.627, 38.372, -61.134]
  MoveL 7262 to (-23.64, 35.16, 106.87) mm, rotated rx 180 ry 0 rz 180 deg; joints [-34.738, -27.023, 99.585, 66.627, 38.372, -61.134]
  Call Extruder(75.36513)
  MoveL 7263 to (-23.15, 35.11, 106.87) mm, rotated rx -180 ry 0 rz 180 deg; joints [-34.671, -26.972, 99.557, 66.602, 38.304, -61.128]
  MoveL 7264 to (-23.15, 35.11, 106.87) mm, rotated rx -180 ry 0 rz 180 deg; joints [-34.671, -26.972, 99.557, 66.602, 38.304, -61.128]
  Call Extruder(75.65986)
  MoveL 7265 to (-22.56, 35.07, 106.87) mm, rotated rx 180 ry 0 rz 180 deg; joints [-34.592, -26.91, 99.523, 66.573, 38.223, -61.122]
  MoveL 7266 to (-22.56, 35.07, 106.87) mm, rotated rx 180 ry 0 rz 180 deg; joints [-34.592, -26.91, 99.523, 66.573, 38.223, -61.122]
  Call Extruder(75.95326)
  MoveL 7267 to (-21.97, 35.02, 106.87) mm, rotated rx 180 ry 0 rz 180 deg; joints [-34.512, -26.847, 99.489, 66.545, 38.142, -61.116]
  MoveL 7268 to (-21.97, 35.02, 106.87) mm, rotated rx 180 ry 0 rz 180 deg; joints [-34.512, -26.847, 99.489, 66.545, 38.142, -61.116]
  Call Extruder(76.38658)
  MoveL 7269 to (-21.1, 34.98, 106.87) mm, rotated rx 180 ry 0 rz 180 deg; joints [-34.399, -26.752, 99.438, 66.507, 38.026, -61.11]
  MoveL 7270 to (-21.1, 34.98, 106.87) mm, rotated rx 180 ry 0 rz 180 deg; joints [-34.399, -26.752, 99.438, 66.507, 38.026, -61.11]
  Call Extruder(76.95875)
  MoveL 7271 to (-19.94, 34.93, 106.87) mm, rotated rx 180 ry 0 rz 180 deg; joints [-34.253, -26.625, 99.369, 66.46, 37.875, -61.106]
  MoveL 7272 to (-19.94, 34.93, 106.87) mm, rotated rx 180 ry 0 rz 180 deg; joints [-34.253, -26.625, 99.369, 66.46, 37.875, -61.106]
  Call Extruder(77.38658)
  MoveL 7273 to (-19.06, 34.91, 106.87) mm, rotated rx 180 ry 0 rz 180 deg; joints [-34.146, -26.528, 99.315, 66.428, 37.764, -61.106]
  Call Extruder(194.03526)
  MoveL 7274 to (219.06, 34.91, 106.87) mm, rotated rx 180 ry 0 rz 180 deg; joints [-18.248, 5.351, 73.143, 58.827, 21.468, -56.973]
  MoveL 7275 to (219.06, 34.91, 106.87) mm, rotated rx 180 ry 0 rz 180 deg; joints [-18.248, 5.351, 73.143, 58.827, 21.468, -56.973]
  Call Extruder(194.75084)
  MoveL 7276 to (220.52, 34.95, 106.87) mm, rotated rx -180 ry 0 rz 180 deg; joints [-18.199, 5.581, 72.892, 58.708, 21.438, -56.856]
  MoveL 7277 to (220.52, 34.95, 106.87) mm, rotated rx -180 ry 0 rz 180 deg; joints [-18.199, 5.581, 72.892, 58.708, 21.438, -56.856]
  Call Extruder(195.32557)
  MoveL 7278 to (221.68, 35, 106.87) mm, rotated rx 180 ry 0 rz 180 deg; joints [-18.162, 5.765, 72.69, 58.614, 21.416, -56.763]
  MoveL 7279 to (221.68, 35, 106.87) mm, rotated rx 180 ry 0 rz 180 deg; joints [-18.162, 5.765, 72.69, 58.614, 21.416, -56.763]
  Call Extruder(195.61897)
  MoveL 7280 to (222.27, 35.05, 106.87) mm, rotated rx 180 ry 0 rz 180 deg; joints [-18.146, 5.86, 72.586, 58.57, 21.407, -56.719]
  MoveL 7281 to (222.27, 35.05, 106.87) mm, rotated rx 180 ry 0 rz 180 deg; joints [-18.146, 5.86, 72.586, 58.57, 21.407, -56.719]
  Call Extruder(195.91369)
  MoveL 7282 to (222.86, 35.09, 106.87) mm, rotated rx -180 ry 0 rz 180 deg; joints [-18.13, 5.955, 72.481, 58.525, 21.398, -56.674]
  MoveL 7283 to (222.86, 35.09, 106.87) mm, rotated rx -180 ry 0 rz 180 deg; joints [-18.13, 5.955, 72.481, 58.525, 21.398, -56.674]
  Call Extruder(196.20975)
  MoveL 7284 to (223.45, 35.14, 106.87) mm, rotated rx -180 ry 0 rz -180 deg; joints [-18.113, 6.051, 72.376, 58.479, 21.39, -56.629]
  MoveL 7285 to (223.45, 35.14, 106.87) mm, rotated rx -180 ry 0 rz -180 deg; joints [-18.113, 6.051, 72.376, 58.479, 21.39, -56.629]
  Call Extruder(196.40602)
  MoveL 7286 to (223.84, 35.18, 106.87) mm, rotated rx -180 ry 0 rz 180 deg; joints [-18.104, 6.114, 72.307, 58.452, 21.386, -56.601]
  MoveL 7287 to (223.84, 35.18, 106.87) mm, rotated rx -180 ry 0 rz 180 deg; joints [-18.104, 6.114, 72.307, 58.452, 21.386, -56.601]
  Call Extruder(196.60317)
  MoveL 7288 to (224.22, 35.23, 106.87) mm, rotated rx -180 ry 0 rz 180 deg; joints [-18.095, 6.178, 72.236, 58.424, 21.382, -56.573]
  MoveL 7289 to (224.22, 35.23, 106.87) mm, rotated rx -180 ry 0 rz 180 deg; joints [-18.095, 6.178, 72.236, 58.424, 21.382, -56.573]
  Call Extruder(196.80118)
  MoveL 7290 to (224.61, 35.27, 106.87) mm, rotated rx 180 ry 0 rz 180 deg; joints [-18.087, 6.241, 72.166, 58.396, 21.378, -56.545]
  MoveL 7291 to (224.61, 35.27, 106.87) mm, rotated rx 180 ry 0 rz 180 deg; joints [-18.087, 6.241, 72.166, 58.396, 21.378, -56.545]
  Call Extruder(197.00005)
  MoveL 7292 to (225, 35.32, 106.87) mm, rotated rx 180 ry 0 rz -180 deg; joints [-18.078, 6.305, 72.096, 58.368, 21.374, -56.517]
  MoveL 7293 to (225, 35.32, 106.87) mm, rotated rx 180 ry 0 rz -180 deg; joints [-18.078, 6.305, 72.096, 58.368, 21.374, -56.517]
  Call Extruder(197.17913)
  MoveL 7294 to (225.34, 35.37, 106.87) mm, rotated rx 180 ry 0 rz 180 deg; joints [-18.07, 6.362, 72.033, 58.344, 21.371, -56.492]
  MoveL 7295 to (225.34, 35.37, 106.87) mm, rotated rx 180 ry 0 rz 180 deg; joints [-18.07, 6.362, 72.033, 58.344, 21.371, -56.492]
  Call Extruder(197.33831)
  MoveL 7296 to (225.65, 35.42, 106.87) mm, rotated rx 180 ry 0 rz 180 deg; joints [-18.065, 6.413, 71.977, 58.323, 21.369, -56.472]
  MoveL 7297 to (225.65, 35.42, 106.87) mm, rotated rx 180 ry 0 rz 180 deg; joints [-18.065, 6.413, 71.977, 58.323, 21.369, -56.472]
  Call Extruder(197.49823)
  MoveL 7298 to (225.96, 35.46, 106.87) mm, rotated rx 180 ry 0 rz 180 deg; joints [-18.059, 6.464, 71.92, 58.303, 21.367, -56.451]
  MoveL 7299 to (225.96, 35.46, 106.87) mm, rotated rx 180 ry 0 rz 180 deg; joints [-18.059, 6.464, 71.92, 58.303, 21.367, -56.451]
  Call Extruder(197.65886)
  MoveL 7300 to (226.26, 35.51, 106.87) mm, rotated rx 180 ry 0 rz 180 deg; joints [-18.054, 6.514, 71.864, 58.282, 21.366, -56.43]
  MoveL 7301 to (226.26, 35.51, 106.87) mm, rotated rx 180 ry 0 rz 180 deg; joints [-18.054, 6.514, 71.864, 58.282, 21.366, -56.43]
  Call Extruder(197.82023)
  MoveL 7302 to (226.57, 35.56, 106.87) mm, rotated rx 180 ry 0 rz -180 deg; joints [-18.048, 6.565, 71.807, 58.262, 21.364, -56.409]
  MoveL 7303 to (226.57, 35.56, 106.87) mm, rotated rx 180 ry 0 rz -180 deg; joints [-18.048, 6.565, 71.807, 58.262, 21.364, -56.409]
  Call Extruder(197.98233)
  MoveL 7304 to (226.87, 35.61, 106.87) mm, rotated rx 180 ry 0 rz 180 deg; joints [-18.042, 6.616, 71.751, 58.241, 21.362, -56.388]
  MoveL 7305 to (226.87, 35.61, 106.87) mm, rotated rx 180 ry 0 rz 180 deg; joints [-18.042, 6.616, 71.751, 58.241, 21.362, -56.388]
  Call Extruder(198.13052)
  MoveL 7306 to (227.15, 35.66, 106.87) mm, rotated rx 180 ry 0 rz 180 deg; joints [-18.038, 6.663, 71.699, 58.223, 21.361, -56.369]
  MoveL 7307 to (227.15, 35.66, 106.87) mm, rotated rx 180 ry 0 rz 180 deg; joints [-18.038, 6.663, 71.699, 58.223, 21.361, -56.369]
  Call Extruder(198.26476)
  MoveL 7308 to (227.4, 35.71, 106.87) mm, rotated rx -180 ry 0 rz 180 deg; joints [-18.034, 6.705, 71.652, 58.207, 21.361, -56.353]
  MoveL 7309 to (227.4, 35.71, 106.87) mm, rotated rx -180 ry 0 rz 180 deg; joints [-18.034, 6.705, 71.652, 58.207, 21.361, -56.353]
  Call Extruder(198.39960)
  MoveL 7310 to (227.65, 35.76, 106.87) mm, rotated rx -180 ry 0 rz -180 deg; joints [-18.031, 6.747, 71.605, 58.192, 21.36, -56.337]
  MoveL 7311 to (227.65, 35.76, 106.87) mm, rotated rx -180 ry 0 rz -180 deg; joints [-18.031, 6.747, 71.605, 58.192, 21.36, -56.337]
  Call Extruder(198.53505)
  MoveL 7312 to (227.9, 35.81, 106.87) mm, rotated rx 180 ry 0 rz 180 deg; joints [-18.027, 6.789, 71.559, 58.176, 21.36, -56.321]
  MoveL 7313 to (227.9, 35.81, 106.87) mm, rotated rx 180 ry 0 rz 180 deg; joints [-18.027, 6.789, 71.559, 58.176, 21.36, -56.321]
  Call Extruder(198.67111)
  MoveL 7314 to (228.15, 35.86, 106.87) mm, rotated rx -180 ry 0 rz 180 deg; joints [-18.024, 6.831, 71.512, 58.16, 21.36, -56.305]
  MoveL 7315 to (228.15, 35.86, 106.87) mm, rotated rx -180 ry 0 rz 180 deg; joints [-18.024, 6.831, 71.512, 58.16, 21.36, -56.305]
  Call Extruder(198.80779)
  MoveL 7316 to (228.4, 35.91, 106.87) mm, rotated rx 180 ry 0 rz -180 deg; joints [-18.02, 6.873, 71.465, 58.144, 21.359, -56.289]
  MoveL 7317 to (228.4, 35.91, 106.87) mm, rotated rx 180 ry 0 rz -180 deg; joints [-18.02, 6.873, 71.465, 58.144, 21.359, -56.289]
  Call Extruder(198.94507)
  MoveL 7318 to (228.64, 35.96, 106.87) mm, rotated rx 180 ry 0 rz 180 deg; joints [-18.017, 6.915, 71.417, 58.128, 21.359, -56.273]
  MoveL 7319 to (228.64, 35.96, 106.87) mm, rotated rx 180 ry 0 rz 180 deg; joints [-18.017, 6.915, 71.417, 58.128, 21.359, -56.273]
  Call Extruder(199.07074)
  MoveL 7320 to (228.87, 36, 106.87) mm, rotated rx 180 ry 0 rz 180 deg; joints [-18.014, 6.954, 71.375, 58.114, 21.359, -56.258]
  MoveL 7321 to (228.87, 36, 106.87) mm, rotated rx 180 ry 0 rz 180 deg; joints [-18.014, 6.954, 71.375, 58.114, 21.359, -56.258]
  Call Extruder(199.18469)
  MoveL 7322 to (229.08, 36.05, 106.87) mm, rotated rx -180 ry 0 rz 180 deg; joints [-18.012, 6.989, 71.336, 58.102, 21.359, -56.245]
  MoveL 7323 to (229.08, 36.05, 106.87) mm, rotated rx -180 ry 0 rz 180 deg; joints [-18.012, 6.989, 71.336, 58.102, 21.359, -56.245]
  Call Extruder(199.29909)
  MoveL 7324 to (229.28, 36.09, 106.87) mm, rotated rx -180 ry 0 rz 180 deg; joints [-18.009, 7.024, 71.297, 58.089, 21.359, -56.232]
  MoveL 7325 to (229.28, 36.09, 106.87) mm, rotated rx -180 ry 0 rz 180 deg; joints [-18.009, 7.024, 71.297, 58.089, 21.359, -56.232]
  Call Extruder(199.41394)
  MoveL 7326 to (229.48, 36.14, 106.87) mm, rotated rx 180 ry 0 rz 180 deg; joints [-18.007, 7.058, 71.258, 58.077, 21.359, -56.219]
  MoveL 7327 to (229.48, 36.14, 106.87) mm, rotated rx 180 ry 0 rz 180 deg; joints [-18.007, 7.058, 71.258, 58.077, 21.359, -56.219]
  Call Extruder(199.52925)
  MoveL 7328 to (229.69, 36.18, 106.87) mm, rotated rx 180 ry 0 rz 180 deg; joints [-18.005, 7.093, 71.219, 58.064, 21.36, -56.206]
  MoveL 7329 to (229.69, 36.18, 106.87) mm, rotated rx 180 ry 0 rz 180 deg; joints [-18.005, 7.093, 71.219, 58.064, 21.36, -56.206]
  Call Extruder(199.65431)
  MoveL 7330 to (229.9, 36.25, 106.87) mm, rotated rx 180 ry 0 rz 180 deg; joints [-18.004, 7.131, 71.176, 58.053, 21.361, -56.195]
  MoveL 7331 to (229.9, 36.25, 106.87) mm, rotated rx 180 ry 0 rz 180 deg; joints [-18.004, 7.131, 71.176, 58.053, 21.361, -56.195]
  Call Extruder(199.77989)
  MoveL 7332 to (230.12, 36.31, 106.87) mm, rotated rx -180 ry 0 rz -180 deg; joints [-18.003, 7.169, 71.134, 58.042, 21.363, -56.183]
  MoveL 7333 to (230.12, 36.31, 106.87) mm, rotated rx -180 ry 0 rz -180 deg; joints [-18.003, 7.169, 71.134, 58.042, 21.363, -56.183]
  Call Extruder(199.90597)
  MoveL 7334 to (230.34, 36.37, 106.87) mm, rotated rx -180 ry 0 rz 180 deg; joints [-18.002, 7.207, 71.092, 58.031, 21.365, -56.171]
  MoveL 7335 to (230.34, 36.37, 106.87) mm, rotated rx -180 ry 0 rz 180 deg; joints [-18.002, 7.207, 71.092, 58.031, 21.365, -56.171]
  Call Extruder(200.01064)
  MoveL 7336 to (230.52, 36.43, 106.87) mm, rotated rx 180 ry 0 rz 180 deg; joints [-18.002, 7.238, 71.056, 58.023, 21.367, -56.162]
  MoveL 7337 to (230.52, 36.43, 106.87) mm, rotated rx 180 ry 0 rz 180 deg; joints [-18.002, 7.238, 71.056, 58.023, 21.367, -56.162]
  Call Extruder(200.11570)
  MoveL 7338 to (230.69, 36.49, 106.87) mm, rotated rx -180 ry 0 rz 180 deg; joints [-18.002, 7.27, 71.021, 58.014, 21.369, -56.153]
  MoveL 7339 to (230.69, 36.49, 106.87) mm, rotated rx -180 ry 0 rz 180 deg; joints [-18.002, 7.27, 71.021, 58.014, 21.369, -56.153]
  Call Extruder(200.22759)
  MoveL 7340 to (230.88, 36.55, 106.87) mm, rotated rx -180 ry 0 rz 180 deg; joints [-18.002, 7.303, 70.984, 58.005, 21.371, -56.144]
  MoveL 7341 to (230.88, 36.55, 106.87) mm, rotated rx -180 ry 0 rz 180 deg; joints [-18.002, 7.303, 70.984, 58.005, 21.371, -56.144]
  Call Extruder(200.33994)
  MoveL 7342 to (231.07, 36.61, 106.87) mm, rotated rx 180 ry 0 rz 180 deg; joints [-18.002, 7.336, 70.946, 57.996, 21.373, -56.134]
  MoveL 7343 to (231.07, 36.61, 106.87) mm, rotated rx 180 ry 0 rz 180 deg; joints [-18.002, 7.336, 70.946, 57.996, 21.373, -56.134]
  Call Extruder(200.45272)
  MoveL 7344 to (231.26, 36.67, 106.87) mm, rotated rx 180 ry 0 rz 180 deg; joints [-18.002, 7.369, 70.909, 57.988, 21.375, -56.125]
  MoveL 7345 to (231.26, 36.67, 106.87) mm, rotated rx 180 ry 0 rz 180 deg; joints [-18.002, 7.369, 70.909, 57.988, 21.375, -56.125]
  Call Extruder(200.56596)
  MoveL 7346 to (231.45, 36.73, 106.87) mm, rotated rx -180 ry 0 rz 180 deg; joints [-18.002, 7.403, 70.872, 57.979, 21.378, -56.115]
  MoveL 7347 to (231.45, 36.73, 106.87) mm, rotated rx -180 ry 0 rz 180 deg; joints [-18.002, 7.403, 70.872, 57.979, 21.378, -56.115]
  Call Extruder(200.67963)
  MoveL 7348 to (231.64, 36.79, 106.87) mm, rotated rx 180 ry 0 rz 180 deg; joints [-18.002, 7.436, 70.834, 57.97, 21.38, -56.105]
  MoveL 7349 to (231.64, 36.79, 106.87) mm, rotated rx 180 ry 0 rz 180 deg; joints [-18.002, 7.436, 70.834, 57.97, 21.38, -56.105]
  Call Extruder(200.86159)
  MoveL 7350 to (231.93, 36.91, 106.87) mm, rotated rx 180 ry 0 rz -180 deg; joints [-18.005, 7.489, 70.774, 57.96, 21.386, -56.094]
  MoveL 7351 to (231.93, 36.91, 106.87) mm, rotated rx 180 ry 0 rz -180 deg; joints [-18.005, 7.489, 70.774, 57.96, 21.386, -56.094]
  Call Extruder(201.04431)
  MoveL 7352 to (232.22, 37.04, 106.87) mm, rotated rx 180 ry 0 rz 180 deg; joints [-18.008, 7.542, 70.715, 57.949, 21.391, -56.082]
  MoveL 7353 to (232.22, 37.04, 106.87) mm, rotated rx 180 ry 0 rz 180 deg; joints [-18.008, 7.542, 70.715, 57.949, 21.391, -56.082]
  Call Extruder(201.21473)
  MoveL 7354 to (232.49, 37.15, 106.87) mm, rotated rx 180 ry 0 rz -180 deg; joints [-18.011, 7.591, 70.659, 57.94, 21.397, -56.072]
  MoveL 7355 to (232.49, 37.15, 106.87) mm, rotated rx 180 ry 0 rz -180 deg; joints [-18.011, 7.591, 70.659, 57.94, 21.397, -56.072]
  Call Extruder(201.37273)
  MoveL 7356 to (232.74, 37.26, 106.87) mm, rotated rx 180 ry 0 rz 180 deg; joints [-18.013, 7.637, 70.608, 57.932, 21.403, -56.062]
  MoveL 7357 to (232.74, 37.26, 106.87) mm, rotated rx 180 ry 0 rz 180 deg; joints [-18.013, 7.637, 70.608, 57.932, 21.403, -56.062]
  Call Extruder(201.53133)
  MoveL 7358 to (232.99, 37.36, 106.87) mm, rotated rx 180 ry 0 rz 180 deg; joints [-18.016, 7.682, 70.556, 57.924, 21.408, -56.053]
  MoveL 7359 to (232.99, 37.36, 106.87) mm, rotated rx 180 ry 0 rz 180 deg; joints [-18.016, 7.682, 70.556, 57.924, 21.408, -56.053]
  Call Extruder(201.73750)
  MoveL 7360 to (233.29, 37.54, 106.87) mm, rotated rx -180 ry 0 rz 180 deg; joints [-18.024, 7.74, 70.491, 57.92, 21.419, -56.047]
  MoveL 7361 to (233.29, 37.54, 106.87) mm, rotated rx -180 ry 0 rz 180 deg; joints [-18.024, 7.74, 70.491, 57.92, 21.419, -56.047]
  Call Extruder(201.94444)
  MoveL 7362 to (233.6, 37.71, 106.87) mm, rotated rx -180 ry 0 rz 180 deg; joints [-18.033, 7.798, 70.425, 57.916, 21.43, -56.041]
  MoveL 7363 to (233.6, 37.71, 106.87) mm, rotated rx -180 ry 0 rz 180 deg; joints [-18.033, 7.798, 70.425, 57.916, 21.43, -56.041]
  Call Extruder(202.15217)
  MoveL 7364 to (233.9, 37.89, 106.87) mm, rotated rx 180 ry 0 rz -180 deg; joints [-18.041, 7.856, 70.36, 57.913, 21.441, -56.035]
  MoveL 7365 to (233.9, 37.89, 106.87) mm, rotated rx 180 ry 0 rz -180 deg; joints [-18.041, 7.856, 70.36, 57.913, 21.441, -56.035]
  Call Extruder(202.36067)
  MoveL 7366 to (234.21, 38.07, 106.87) mm, rotated rx -180 ry 0 rz -180 deg; joints [-18.049, 7.914, 70.294, 57.909, 21.452, -56.029]
  MoveL 7367 to (234.21, 38.07, 106.87) mm, rotated rx -180 ry 0 rz -180 deg; joints [-18.049, 7.914, 70.294, 57.909, 21.452, -56.029]
  Call Extruder(202.54021)
  MoveL 7368 to (234.45, 38.24, 106.87) mm, rotated rx -180 ry 0 rz 180 deg; joints [-18.06, 7.963, 70.239, 57.911, 21.464, -56.029]
  MoveL 7369 to (234.45, 38.24, 106.87) mm, rotated rx -180 ry 0 rz 180 deg; joints [-18.06, 7.963, 70.239, 57.911, 21.464, -56.029]
  Call Extruder(202.87363)
  MoveL 7370 to (234.9, 38.57, 106.87) mm, rotated rx 180 ry 0 rz 180 deg; joints [-18.079, 8.053, 70.137, 57.914, 21.486, -56.029]
  MoveL 7371 to (234.9, 38.57, 106.87) mm, rotated rx 180 ry 0 rz 180 deg; joints [-18.079, 8.053, 70.137, 57.914, 21.486, -56.029]
  Call Extruder(203.20823)
  MoveL 7372 to (235.35, 38.9, 106.87) mm, rotated rx 180 ry 0 rz -180 deg; joints [-18.099, 8.143, 70.035, 57.918, 21.509, -56.028]
  Call Extruder(204.03618)
  MoveL 7373 to (236.39, 39.81, 106.87) mm, rotated rx 180 ry 0 rz -180 deg; joints [-18.16, 8.358, 69.789, 57.948, 21.576, -56.047]
  Call Extruder(204.86412)
  MoveL 7374 to (237.3, 40.85, 106.87) mm, rotated rx -180 ry 0 rz 180 deg; joints [-18.24, 8.561, 69.558, 58.006, 21.657, -56.092]
  Call Extruder(205.03142)
  MoveL 7375 to (237.47, 41.07, 106.87) mm, rotated rx 180 ry 0 rz -180 deg; joints [-18.258, 8.6, 69.514, 58.022, 21.675, -56.105]
  MoveL 7376 to (237.47, 41.07, 106.87) mm, rotated rx 180 ry 0 rz -180 deg; joints [-18.258, 8.6, 69.514, 58.022, 21.675, -56.105]
  Call Extruder(205.36483)
  MoveL 7377 to (237.79, 41.52, 106.87) mm, rotated rx -180 ry 0 rz 180 deg; joints [-18.295, 8.677, 69.425, 58.053, 21.712, -56.131]
  MoveL 7378 to (237.79, 41.52, 106.87) mm, rotated rx -180 ry 0 rz 180 deg; joints [-18.295, 8.677, 69.425, 58.053, 21.712, -56.131]
  Call Extruder(205.69706)
  MoveL 7379 to (238.12, 41.97, 106.87) mm, rotated rx -180 ry 0 rz 180 deg; joints [-18.332, 8.754, 69.337, 58.085, 21.748, -56.156]
  MoveL 7380 to (238.12, 41.97, 106.87) mm, rotated rx -180 ry 0 rz 180 deg; joints [-18.332, 8.754, 69.337, 58.085, 21.748, -56.156]
  Call Extruder(205.81476)
  MoveL 7381 to (238.22, 42.15, 106.87) mm, rotated rx -180 ry 0 rz 180 deg; joints [-18.346, 8.78, 69.308, 58.099, 21.763, -56.168]
  MoveL 7382 to (238.22, 42.15, 106.87) mm, rotated rx -180 ry 0 rz 180 deg; joints [-18.346, 8.78, 69.308, 58.099, 21.763, -56.168]
  Call Extruder(206.02249)
  MoveL 7383 to (238.4, 42.45, 106.87) mm, rotated rx -180 ry 0 rz 180 deg; joints [-18.373, 8.825, 69.256, 58.124, 21.788, -56.19]
  MoveL 7384 to (238.4, 42.45, 106.87) mm, rotated rx -180 ry 0 rz 180 deg; joints [-18.373, 8.825, 69.256, 58.124, 21.788, -56.19]
  Call Extruder(206.22943)
  MoveL 7385 to (238.57, 42.75, 106.87) mm, rotated rx 180 ry 0 rz 180 deg; joints [-18.399, 8.869, 69.205, 58.149, 21.813, -56.211]
  MoveL 7386 to (238.57, 42.75, 106.87) mm, rotated rx 180 ry 0 rz 180 deg; joints [-18.399, 8.869, 69.205, 58.149, 21.813, -56.211]
  Call Extruder(206.43560)
  MoveL 7387 to (238.75, 43.06, 106.87) mm, rotated rx -180 ry 0 rz 180 deg; joints [-18.425, 8.914, 69.153, 58.174, 21.839, -56.232]
  MoveL 7388 to (238.75, 43.06, 106.87) mm, rotated rx -180 ry 0 rz 180 deg; joints [-18.425, 8.914, 69.153, 58.174, 21.839, -56.232]
  Call Extruder(206.61728)
  MoveL 7389 to (238.89, 43.34, 106.87) mm, rotated rx -180 ry 0 rz -180 deg; joints [-18.45, 8.952, 69.109, 58.199, 21.862, -56.253]
  MoveL 7390 to (238.89, 43.34, 106.87) mm, rotated rx -180 ry 0 rz -180 deg; joints [-18.45, 8.952, 69.109, 58.199, 21.862, -56.253]
  Call Extruder(206.77529)
  MoveL 7391 to (239, 43.58, 106.87) mm, rotated rx 180 ry 0 rz 180 deg; joints [-18.472, 8.983, 69.074, 58.223, 21.883, -56.274]
  MoveL 7392 to (239, 43.58, 106.87) mm, rotated rx 180 ry 0 rz 180 deg; joints [-18.472, 8.983, 69.074, 58.223, 21.883, -56.274]
  Call Extruder(206.93270)
  MoveL 7393 to (239.11, 43.83, 106.87) mm, rotated rx -180 ry 0 rz 180 deg; joints [-18.495, 9.014, 69.038, 58.247, 21.905, -56.295]
  MoveL 7394 to (239.11, 43.83, 106.87) mm, rotated rx -180 ry 0 rz 180 deg; joints [-18.495, 9.014, 69.038, 58.247, 21.905, -56.295]
  Call Extruder(207.11542)
  MoveL 7395 to (239.22, 44.13, 106.87) mm, rotated rx 180 ry 0 rz 180 deg; joints [-18.522, 9.049, 68.997, 58.275, 21.93, -56.319]
  MoveL 7396 to (239.22, 44.13, 106.87) mm, rotated rx 180 ry 0 rz 180 deg; joints [-18.522, 9.049, 68.997, 58.275, 21.93, -56.319]
  Call Extruder(207.29737)
  MoveL 7397 to (239.35, 44.42, 106.87) mm, rotated rx -180 ry 0 rz -180 deg; joints [-18.549, 9.085, 68.956, 58.304, 21.955, -56.344]
  MoveL 7398 to (239.35, 44.42, 106.87) mm, rotated rx -180 ry 0 rz -180 deg; joints [-18.549, 9.085, 68.956, 58.304, 21.955, -56.344]
  Call Extruder(207.44470)
  MoveL 7399 to (239.44, 44.66, 106.87) mm, rotated rx 180 ry 0 rz 180 deg; joints [-18.571, 9.113, 68.924, 58.328, 21.976, -56.365]
  MoveL 7400 to (239.44, 44.66, 106.87) mm, rotated rx 180 ry 0 rz 180 deg; joints [-18.571, 9.113, 68.924, 58.328, 21.976, -56.365]
  Call Extruder(207.55794)
  MoveL 7401 to (239.5, 44.85, 106.87) mm, rotated rx 180 ry 0 rz 180 deg; joints [-18.589, 9.133, 68.901, 58.348, 21.992, -56.382]
  MoveL 7402 to (239.5, 44.85, 106.87) mm, rotated rx 180 ry 0 rz 180 deg; joints [-18.589, 9.133, 68.901, 58.348, 21.992, -56.382]
  Call Extruder(207.67073)
  MoveL 7403 to (239.56, 45.03, 106.87) mm, rotated rx 180 ry 0 rz 180 deg; joints [-18.607, 9.153, 68.877, 58.367, 22.009, -56.4]
  MoveL 7404 to (239.56, 45.03, 106.87) mm, rotated rx 180 ry 0 rz 180 deg; joints [-18.607, 9.153, 68.877, 58.367, 22.009, -56.4]
  Call Extruder(207.78308)
  MoveL 7405 to (239.62, 45.22, 106.87) mm, rotated rx -180 ry 0 rz 180 deg; joints [-18.625, 9.174, 68.854, 58.387, 22.025, -56.417]
  MoveL 7406 to (239.62, 45.22, 106.87) mm, rotated rx -180 ry 0 rz 180 deg; joints [-18.625, 9.174, 68.854, 58.387, 22.025, -56.417]
  Call Extruder(207.89498)
  MoveL 7407 to (239.68, 45.41, 106.87) mm, rotated rx -180 ry 0 rz -180 deg; joints [-18.642, 9.194, 68.831, 58.407, 22.042, -56.434]
  MoveL 7408 to (239.68, 45.41, 106.87) mm, rotated rx -180 ry 0 rz -180 deg; joints [-18.642, 9.194, 68.831, 58.407, 22.042, -56.434]
  Call Extruder(208.01638)
  MoveL 7409 to (239.75, 45.62, 106.87) mm, rotated rx 180 ry 0 rz -180 deg; joints [-18.662, 9.216, 68.805, 58.429, 22.06, -56.453]
  MoveL 7410 to (239.75, 45.62, 106.87) mm, rotated rx 180 ry 0 rz -180 deg; joints [-18.662, 9.216, 68.805, 58.429, 22.06, -56.453]
  Call Extruder(208.14717)
  MoveL 7411 to (239.81, 45.84, 106.87) mm, rotated rx 180 ry 0 rz 180 deg; joints [-18.683, 9.239, 68.778, 58.452, 22.08, -56.474]
  MoveL 7412 to (239.81, 45.84, 106.87) mm, rotated rx 180 ry 0 rz 180 deg; joints [-18.683, 9.239, 68.778, 58.452, 22.08, -56.474]
  Call Extruder(208.27740)
  MoveL 7413 to (239.88, 46.06, 106.87) mm, rotated rx -180 ry 0 rz -180 deg; joints [-18.705, 9.262, 68.752, 58.476, 22.099, -56.495]
  MoveL 7414 to (239.88, 46.06, 106.87) mm, rotated rx -180 ry 0 rz -180 deg; joints [-18.705, 9.262, 68.752, 58.476, 22.099, -56.495]
  Call Extruder(208.40706)
  MoveL 7415 to (239.95, 46.29, 106.87) mm, rotated rx -180 ry 0 rz 180 deg; joints [-18.726, 9.286, 68.725, 58.5, 22.119, -56.516]
  MoveL 7416 to (239.95, 46.29, 106.87) mm, rotated rx -180 ry 0 rz 180 deg; joints [-18.726, 9.286, 68.725, 58.5, 22.119, -56.516]
  Call Extruder(208.53615)
  MoveL 7417 to (240.02, 46.51, 106.87) mm, rotated rx 180 ry 0 rz 180 deg; joints [-18.747, 9.309, 68.698, 58.523, 22.139, -56.536]
  MoveL 7418 to (240.02, 46.51, 106.87) mm, rotated rx 180 ry 0 rz 180 deg; joints [-18.747, 9.309, 68.698, 58.523, 22.139, -56.536]
  Call Extruder(208.65121)
  MoveL 7419 to (240.06, 46.72, 106.87) mm, rotated rx 180 ry 0 rz 180 deg; joints [-18.767, 9.328, 68.676, 58.546, 22.157, -56.557]
  MoveL 7420 to (240.06, 46.72, 106.87) mm, rotated rx 180 ry 0 rz 180 deg; joints [-18.767, 9.328, 68.676, 58.546, 22.157, -56.557]
  Call Extruder(208.76581)
  MoveL 7421 to (240.11, 46.92, 106.87) mm, rotated rx -180 ry 0 rz 180 deg; joints [-18.787, 9.346, 68.655, 58.57, 22.175, -56.577]
  MoveL 7422 to (240.11, 46.92, 106.87) mm, rotated rx -180 ry 0 rz 180 deg; joints [-18.787, 9.346, 68.655, 58.57, 22.175, -56.577]
  Call Extruder(208.87996)
  MoveL 7423 to (240.15, 47.12, 106.87) mm, rotated rx 180 ry 0 rz 180 deg; joints [-18.807, 9.365, 68.633, 58.593, 22.193, -56.598]
  MoveL 7424 to (240.15, 47.12, 106.87) mm, rotated rx 180 ry 0 rz 180 deg; joints [-18.807, 9.365, 68.633, 58.593, 22.193, -56.598]
  Call Extruder(208.99365)
  MoveL 7425 to (240.2, 47.33, 106.87) mm, rotated rx 180 ry 0 rz 180 deg; joints [-18.827, 9.384, 68.612, 58.616, 22.212, -56.618]
  MoveL 7426 to (240.2, 47.33, 106.87) mm, rotated rx 180 ry 0 rz 180 deg; joints [-18.827, 9.384, 68.612, 58.616, 22.212, -56.618]
  Call Extruder(209.11906)
  MoveL 7427 to (240.24, 47.56, 106.87) mm, rotated rx 180 ry 0 rz 180 deg; joints [-18.85, 9.404, 68.588, 58.641, 22.232, -56.641]
  MoveL 7428 to (240.24, 47.56, 106.87) mm, rotated rx 180 ry 0 rz 180 deg; joints [-18.85, 9.404, 68.588, 58.641, 22.232, -56.641]
  Call Extruder(209.25604)
  MoveL 7429 to (240.29, 47.8, 106.87) mm, rotated rx 180 ry 0 rz 180 deg; joints [-18.874, 9.426, 68.563, 58.67, 22.254, -56.666]
  MoveL 7430 to (240.29, 47.8, 106.87) mm, rotated rx 180 ry 0 rz 180 deg; joints [-18.874, 9.426, 68.563, 58.67, 22.254, -56.666]
  Call Extruder(209.39241)
  MoveL 7431 to (240.34, 48.05, 106.87) mm, rotated rx -180 ry 0 rz 180 deg; joints [-18.899, 9.448, 68.537, 58.698, 22.276, -56.691]
  MoveL 7432 to (240.34, 48.05, 106.87) mm, rotated rx -180 ry 0 rz 180 deg; joints [-18.899, 9.448, 68.537, 58.698, 22.276, -56.691]
  Call Extruder(209.52817)
  MoveL 7433 to (240.39, 48.3, 106.87) mm, rotated rx -180 ry 0 rz -180 deg; joints [-18.923, 9.47, 68.512, 58.727, 22.299, -56.716]
  MoveL 7434 to (240.39, 48.3, 106.87) mm, rotated rx -180 ry 0 rz -180 deg; joints [-18.923, 9.47, 68.512, 58.727, 22.299, -56.716]
  Call Extruder(209.66331)
  MoveL 7435 to (240.44, 48.55, 106.87) mm, rotated rx 180 ry 0 rz 180 deg; joints [-18.948, 9.492, 68.486, 58.755, 22.321, -56.741]
  MoveL 7436 to (240.44, 48.55, 106.87) mm, rotated rx 180 ry 0 rz 180 deg; joints [-18.948, 9.492, 68.486, 58.755, 22.321, -56.741]
  Call Extruder(209.79785)
  MoveL 7437 to (240.49, 48.8, 106.87) mm, rotated rx -180 ry 0 rz -180 deg; joints [-18.973, 9.514, 68.461, 58.783, 22.344, -56.766]
  MoveL 7438 to (240.49, 48.8, 106.87) mm, rotated rx -180 ry 0 rz -180 deg; joints [-18.973, 9.514, 68.461, 58.783, 22.344, -56.766]
  Call Extruder(209.93178)
  MoveL 7439 to (240.54, 49.05, 106.87) mm, rotated rx -180 ry 0 rz 180 deg; joints [-18.997, 9.536, 68.435, 58.811, 22.366, -56.791]
  MoveL 7440 to (240.54, 49.05, 106.87) mm, rotated rx -180 ry 0 rz 180 deg; joints [-18.997, 9.536, 68.435, 58.811, 22.366, -56.791]
  Call Extruder(210.07964)
  MoveL 7441 to (240.59, 49.33, 106.87) mm, rotated rx 180 ry 0 rz 180 deg; joints [-19.025, 9.559, 68.408, 58.842, 22.391, -56.819]
  MoveL 7442 to (240.59, 49.33, 106.87) mm, rotated rx 180 ry 0 rz 180 deg; joints [-19.025, 9.559, 68.408, 58.842, 22.391, -56.819]
  Call Extruder(210.24139)
  MoveL 7443 to (240.64, 49.63, 106.87) mm, rotated rx 180 ry 0 rz 180 deg; joints [-19.055, 9.584, 68.379, 58.878, 22.418, -56.85]
  MoveL 7444 to (240.64, 49.63, 106.87) mm, rotated rx 180 ry 0 rz 180 deg; joints [-19.055, 9.584, 68.379, 58.878, 22.418, -56.85]
  Call Extruder(210.40241)
  MoveL 7445 to (240.69, 49.94, 106.87) mm, rotated rx 180 ry 0 rz 180 deg; joints [-19.086, 9.609, 68.35, 58.913, 22.446, -56.882]
  MoveL 7446 to (240.69, 49.94, 106.87) mm, rotated rx 180 ry 0 rz 180 deg; joints [-19.086, 9.609, 68.35, 58.913, 22.446, -56.882]
  Call Extruder(210.56270)
  MoveL 7447 to (240.73, 50.24, 106.87) mm, rotated rx 180 ry 0 rz 180 deg; joints [-19.116, 9.635, 68.32, 58.948, 22.474, -56.913]
  MoveL 7448 to (240.73, 50.24, 106.87) mm, rotated rx 180 ry 0 rz 180 deg; joints [-19.116, 9.635, 68.32, 58.948, 22.474, -56.913]
  Call Extruder(210.72226)
  MoveL 7449 to (240.78, 50.55, 106.87) mm, rotated rx 180 ry 0 rz 180 deg; joints [-19.146, 9.66, 68.291, 58.983, 22.501, -56.944]
  MoveL 7450 to (240.78, 50.55, 106.87) mm, rotated rx 180 ry 0 rz 180 deg; joints [-19.146, 9.66, 68.291, 58.983, 22.501, -56.944]
  Call Extruder(210.88109)
  MoveL 7451 to (240.83, 50.86, 106.87) mm, rotated rx -180 ry 0 rz -180 deg; joints [-19.177, 9.685, 68.262, 59.018, 22.529, -56.975]
  MoveL 7452 to (240.83, 50.86, 106.87) mm, rotated rx -180 ry 0 rz -180 deg; joints [-19.177, 9.685, 68.262, 59.018, 22.529, -56.975]
  Call Extruder(211.05976)
  MoveL 7453 to (240.88, 51.2, 106.87) mm, rotated rx -180 ry 0 rz 180 deg; joints [-19.212, 9.712, 68.23, 59.058, 22.56, -57.01]
  MoveL 7454 to (240.88, 51.2, 106.87) mm, rotated rx -180 ry 0 rz 180 deg; joints [-19.212, 9.712, 68.23, 59.058, 22.56, -57.01]
  Call Extruder(211.25821)
  MoveL 7455 to (240.92, 51.59, 106.87) mm, rotated rx 180 ry 0 rz 180 deg; joints [-19.251, 9.742, 68.195, 59.104, 22.596, -57.051]
